// SIMATIC STEP 7 (V5.x) project L38_X52_EC1
// CPU: CPU
// station: P_ADR_BUS
// station: Matériel
// station: API
// station: P_ADR_BUS
// station: Configuration
// station: MOP
// program: PROG
// program: Programa S7_back

SYMBOL_TABLE
"IBD"	DB 95	DB 95	// FACILITY: DATA BASE DB / DB BASE DE DONNEE
"IIT"	DB 96	DB 96	// FACILITY: PART TABLE / DB TABLE PIECE
END_SYMBOL_TABLE

DATA_BLOCK "IBD"	// DB 95
TITLE = FACILITY: DATABASE DB CONTROL
NAME : IBD
VERSION : 0.1
  STRUCT
   BDD : ARRAY  [1 .. 8, 1 .. 200 ] OF WORD ;	//SPARE
  END_STRUCT ;	
BEGIN
END_DATA_BLOCK

DATA_BLOCK "IIT"	// DB 96
TITLE = FACILITY: PART WORD TABLE
NAME : IIT
VERSION : 1.0
  STRUCT
   A0 : STRUCT 	//PART WORD A0
    MP : STRUCT 	//PART MEMORY / MOT PIECE
     MPP : BOOL ;	//PRESENT PART MEMORY / MEMOIRE PIECE PRESENTE
     MPAT : BOOL ;	//PART WITH WORK MEMORY / MEMOIRE PIECE A TRAVAILLER
     MPST : BOOL ;	//PART WITHOUT WORK MEMORY / MEMOIRE PIECE SANS TRAVAIL
     MPAM : BOOL ;	//PART MEMORY TO MATCH / MEMOIRE PIECE A MARIER
     MPAE : BOOL ;	//PART MEMORY TO EVACUATE / MEMOIRE PIECE A EVACUER
     MPP1 : BOOL ;	//INTERMEDIATE PRESENT PART MEMORY / MEMOIRE PIECE PRESENTE INTERMEDIAIRE
     MPP2 : BOOL ;	//INTERMEDIATE PRESENT PART MEMORY / MEMOIRE PIECE PRESENTE INTERMEDIAIRE
     MPP3 : BOOL ;	//INTERMEDIATE PRESENT PART MEMORY / MEMOIRE PIECE PRESENTE INTERMEDIAIRE
     MPP4 : BOOL ;	//INTERMEDIATE PRESENT PART MEMORY / MEMOIRE PIECE PRESENTE INTERMEDIAIRE
     MPP5 : BOOL ;	//INTERMEDIATE PRESENT PART MEMORY / MEMOIRE PIECE PRESENTE INTERMEDIAIRE
     MPP6 : BOOL ;	//INTERMEDIATE PRESENT PART MEMORY / MEMOIRE PIECE PRESENTE INTERMEDIAIRE
     MPP7 : BOOL ;	//INTERMEDIATE PRESENT PART MEMORY / MEMOIRE PIECE PRESENTE INTERMEDIAIRE
     MPP8 : BOOL ;	//INTERMEDIATE PRESENT PART MEMORY / MEMOIRE PIECE PRESENTE INTERMEDIAIRE
     MPT : BOOL ;	//PART COMPLETE MEMORY / MEMOIRE PIECE TRAVAILLE
     MPLNOK : BOOL ;	//LAUCHING PART MEMORY NOK / MEMOIRE LANCEMENT PIECE NON OK
     MPLNOR : BOOL ;	//LAUCHING PART MEMORY OK / MEMOIRE LANCEMENT PIECE OK
    END_STRUCT ;
    MS : STRUCT 	//SUPPORT WORD / MOT SUPPORT
     MSP : BOOL ;	//SUPPORT PRESENCE MEMORY / MEMOIRE SUPPORT PRESENT
     MSAE : BOOL ;	//SUPPORT TO EVACUATE MEMORY / MEMOIRE SUPPORT A EVACUER
     MSEBD : BOOL ;	//WRITING DATABASE SUPPORT MEMORY / MEMOIRE SUPPORT ECRITURE BASE DE DONNEE
     MSMBD : BOOL ;	//MODIFICATION DATABASE SUPPORT MEMORY / MEMOIRE SUPPORT MODIF BASE DE DONNEE
     MSLBD : BOOL ;	//READING DATABASE SUPPORT MEMORY / MEMOIRE SUPPORT LECTURE BASE DE DONNEE
     MSAP : BOOL ;	//PASSAGE AUTHORIZATION SUPPORT MEMORY / MEMOIRE SUPPORT AUTORISATION DE PASSAGE
     MRCPF : BOOL ;	//PART TO DO PROCESS CODE SEARCH MEMORY / MEMOIRE RECH CODES PROCESS A FAIRE
     MRCPS : BOOL ;	//NEXT PART PROCESS CODE SEARCH MEMORY / MEMOIRE RECH CODES PROCESS SUIVANT
     MSLRFID : BOOL ;	//READING RFID SUPPORT MEMORY / MEMOIRE SUPPORT LECTURE RFID
     MSERFID : BOOL ;	//WRITING RFID SUPPORT MEMORY / MEMOIRE SUPPORT ECRITURE RFID
     RES1 : BOOL ;	//SPARE / RESERVE
     RES2 : BOOL ;	//SPARE / RESERVE
     RES3 : BOOL ;	//SPARE / RESERVE
     RES4 : BOOL ;	//SPARE / RESERVE
     RES5 : BOOL ;	//SPARE / RESERVE
     MSLHS : BOOL ;	//LOCAL PRODUCTION MEMORY SUPPORT / MEMOIRE SUPPORT LANCE HORS SIPTOL
    END_STRUCT ;
    NSUP : INT ;	//SUPPORT NUMBER / NUMERO DE SUPPORT
    NFILM : INT ;	//FILM NUMBER / NUMERO DE FILM
    NORDRE : INT ;	//ORDER NUMBER / NUMERO D ORDRE
    CDIV1 : INT ;	//FAMILIA / FAMILLE (CDIV1)
    CDIV2 : INT ;	//FASE / PHASE (CDIV2)
    CDIV3 : INT ;	//MODELO / MODELE (CDIV3)
    CDIV4 : INT ;	//TECHO (CDIV4)
    CDIV5 : INT ;	//VERSION (CDIV5)
    DESFI : INT ;	//FINAL DISPATCH / DESTINATION FINALE
    CSORT : INT ;	//CAUSE DE SORTIE
    DAT : STRUCT 	//DEFINITION / ATTENTE TRAVAIL
     B8 : BOOL ;	//PALETTE DE VIDAGE PERIMETRE (HORS SIPTOL)
     B9 : BOOL ;	//DEVERMINAGE PIECE / PALETTE (HORS SIPTOL)
     B10 : BOOL ;	//PALETTE DE MAP(HORS SIPTOL)
     B11 : BOOL ;	//PALETTE DE CHANGEMENT ELECTRODE BR (HORS SIPTOL)
     B12 : BOOL ;	//PALETTE DE CHANGEMENT ELECTRODE CS (HORS SIPTOL)
     B13 : BOOL ;	//DEVERMINAGE PIECE / PALETTE (AVEC SIPTOL)
     B14 : BOOL ;
     B15 : BOOL ;
     FABSPF : BOOL ;	//0 = AVEC TRAVAIL / 1 = SANS TRAVAIL (P1)
     B1 : BOOL ;
     B2 : BOOL ;	//0 = SUPPORT PLEIN / 1 = SUPPORT VIDE
     B3 : BOOL ;
     B4 : BOOL ;
     B5 : BOOL ;
     B6 : BOOL ;
     B7 : BOOL ;
    END_STRUCT ;
    CRAPI : STRUCT 	//PLC DISPATCHING REASON / CAUSE ROUTAGE API
     B8 : BOOL ;
     B9 : BOOL ;
     B10 : BOOL ;
     B11 : BOOL ;
     B12 : BOOL ;
     B13 : BOOL ;
     B14 : BOOL ;
     B15 : BOOL ;
     B0 : BOOL ;
     B1 : BOOL ;
     B2 : BOOL ;
     RARET : BOOL ;	//PIECE ANALYSE - RETOUCHE
     B4 : BOOL ;
     B5 : BOOL ;
     B6 : BOOL ;
     B7 : BOOL ;
    END_STRUCT ;
    MGEST : STRUCT 	//MOT DE GESTION RECALAGE
     MPFNOR : BOOL ;	//MEMOIRE PIECE FLUX NORMAL
     MPSTC : BOOL ;	//MEMOIRE PIECE A SORTIR TOUS CAS
     MPSOR : BOOL ;	//MEMOIRE PIECE A SORTIR (SORTIE SIPTOL BONNE)
     MPSSU : BOOL ;	//MEMOIRE PIECE A SORTIR (SUBTITUTION PIECE BONNE)
     MPSDI : BOOL ;	//MEMOIRE PIECE A SORTIR (DISCORDANCE)
     MPSSUL : BOOL ;	//MEMOIRE PIECE A SORTIR (SUBTITUTION PIECE LOUPEE)
     MPSL : BOOL ;	//MEMOIRE PIECE A SORTIR (SORTIE LOUPEE)
     MPSF99 : BOOL ;	//MEMOIRE PIECE A SORTIR (MAP FILM 99)
     MPETC : BOOL ;	//MEMOIRE PIECE A ENTRER TOUTS CAS
     MPEOR : BOOL ;	//MEMOIRE PIECE EN ENTREE (DEMANDE SIPTOL)
     MPESUB : BOOL ;	//MEMOIRE PIECE EN ENTREE (SUBTITUTION PIECE BONNE)
     MPEDI : BOOL ;	//MEMOIRE PIECE EN ENTREE (DISCORDANCE)
     MPESUL : BOOL ;	//MEMOIRE PIECE EN ENTREE (SUBTITUTION PIECE LOUPEE)
     MPOCV : BOOL ;	//MEMOIRE PIECE A SORTIR VEHICULE ANNULE + CROCHET VIDE
     MESUTC : BOOL ;	//MEMOIRE EN ENTREE SUBSTITUTION TOUS CAS (PIECE BONNE OU MAUVAISE)
     MSSUTC : BOOL ;	//MEMOIRE SORTIE SUBSTITUTION TOUS CAS (PIECE BONNE OU MAUVAISE)
    END_STRUCT ;
    TVEH : STRUCT 	//TYPO DE VEHICULO
     B8 : BOOL ;
     B9 : BOOL ;
     B10 : BOOL ;
     B11 : BOOL ;
     B12 : BOOL ;
     B13 : BOOL ;
     B14 : BOOL ;
     FABSPF : BOOL ;	//FABRICATION SANS PIECE AU FILM
     SPE : BOOL ;	//UNIT ESPECIAL
     B1 : BOOL ;
     B2 : BOOL ;
     B3 : BOOL ;
     B4 : BOOL ;
     B5 : BOOL ;
     B6 : BOOL ;
     B7 : BOOL ;
    END_STRUCT ;
    SPARE : ARRAY  [1 .. 4 ] OF INT ;	//SPARE
   END_STRUCT ;
   A0_TT : STRUCT 	//WORK TABLE A0
    MFT : STRUCT 	//END OF WORK MEMORY
     MFT1 : BOOL ;	//END OF WORK MEMORY 1 - SPARE
     MFT2 : BOOL ;	//END OF WORK MEMORY 2 - SPARE
     MFT3 : BOOL ;	//END OF WORK MEMORY 3 - SPARE
     MFT4 : BOOL ;	//END OF WORK MEMORY 4 - SPARE
     MFT5 : BOOL ;	//END OF WORK MEMORY 5 - SPARE
     MFT6 : BOOL ;	//END OF WORK MEMORY 6 - SPARE
     MFT7 : BOOL ;	//END OF WORK MEMORY 7 - SPARE
     MFT8 : BOOL ;	//END OF WORK MEMORY 8 - SPARE
     MFT9 : BOOL ;	//END OF WORK MEMORY 9 - SPARE
     MFT10 : BOOL ;	//END OF WORK MEMORY 10 - SPARE
     MFT11 : BOOL ;	//END OF WORK MEMORY 11 - SPARE
     MFT12 : BOOL ;	//END OF WORK MEMORY 12 - SPARE
     MFT13 : BOOL ;	//END OF WORK MEMORY 13 - SPARE
     MFT14 : BOOL ;	//END OF WORK MEMORY 14 - SPARE
     MFT15 : BOOL ;	//END OF WORK MEMORY 15 - SPARE
     MFT16 : BOOL ;	//END OF WORK MEMORY 16 - SPARE
    END_STRUCT ;
    A1 : STRUCT 	//END OF WORK MEMORY A1
     MFT1 : BOOL ;	//END OF WORK MEMORY 1 - SPARE
     MFT2 : BOOL ;	//END OF WORK MEMORY 2 - SPARE
     MFT3 : BOOL ;	//END OF WORK MEMORY 3 - SPARE
     MFT4 : BOOL ;	//END OF WORK MEMORY 4 - SPARE
     MFT5 : BOOL ;	//END OF WORK MEMORY 5 - SPARE
     MFT6 : BOOL ;	//END OF WORK MEMORY 6 - SPARE
     MFT7 : BOOL ;	//END OF WORK MEMORY 7 - SPARE
     MFT8 : BOOL ;	//END OF WORK MEMORY 8 - SPARE
    END_STRUCT ;
    A2 : STRUCT 	//END OF WORK MEMORY A2
     MFT1 : BOOL ;	//END OF WORK MEMORY 1 - SPARE
     MFT2 : BOOL ;	//END OF WORK MEMORY 2 - SPARE
     MFT3 : BOOL ;	//END OF WORK MEMORY 3 - SPARE
     MFT4 : BOOL ;	//END OF WORK MEMORY 4 - SPARE
     MFT5 : BOOL ;	//END OF WORK MEMORY 5 - SPARE
     MFT6 : BOOL ;	//END OF WORK MEMORY 6 - SPARE
     MFT7 : BOOL ;	//END OF WORK MEMORY 7 - SPARE
     MFT8 : BOOL ;	//END OF WORK MEMORY 8 - SPARE
    END_STRUCT ;
    A3 : STRUCT 	//END OF WORK MEMORY A3
     MFT1 : BOOL ;	//END OF WORK MEMORY 1 - SPARE
     MFT2 : BOOL ;	//END OF WORK MEMORY 2 - SPARE
     MFT3 : BOOL ;	//END OF WORK MEMORY 3 - SPARE
     MFT4 : BOOL ;	//END OF WORK MEMORY 4 - SPARE
     MFT5 : BOOL ;	//END OF WORK MEMORY 5 - SPARE
     MFT6 : BOOL ;	//END OF WORK MEMORY 6 - SPARE
     MFT7 : BOOL ;	//END OF WORK MEMORY 7 - SPARE
     MFT8 : BOOL ;	//END OF WORK MEMORY 8 - SPARE
    END_STRUCT ;
    SPARE : ARRAY  [1 .. 16 ] OF INT ;	//SPARE
   END_STRUCT ;
   A0w : STRUCT 	//PART WORD A0w
    MP : STRUCT 	//PART MEMORY / MOT PIECE
     MPP : BOOL ;	//PRESENT PART MEMORY / MEMOIRE PIECE PRESENTE
     MPAT : BOOL ;	//PART WITH WORK MEMORY / MEMOIRE PIECE A TRAVAILLER
     MPST : BOOL ;	//PART WITHOUT WORK MEMORY / MEMOIRE PIECE SANS TRAVAIL
     MPAM : BOOL ;	//PART MEMORY TO MATCH / MEMOIRE PIECE A MARIER
     MPAE : BOOL ;	//PART MEMORY TO EVACUATE / MEMOIRE PIECE A EVACUER
     MPP1 : BOOL ;	//INTERMEDIATE PRESENT PART MEMORY / MEMOIRE PIECE PRESENTE INTERMEDIAIRE
     MPP2 : BOOL ;	//INTERMEDIATE PRESENT PART MEMORY / MEMOIRE PIECE PRESENTE INTERMEDIAIRE
     MPP3 : BOOL ;	//INTERMEDIATE PRESENT PART MEMORY / MEMOIRE PIECE PRESENTE INTERMEDIAIRE
     MPP4 : BOOL ;	//INTERMEDIATE PRESENT PART MEMORY / MEMOIRE PIECE PRESENTE INTERMEDIAIRE
     MPP5 : BOOL ;	//INTERMEDIATE PRESENT PART MEMORY / MEMOIRE PIECE PRESENTE INTERMEDIAIRE
     MPP6 : BOOL ;	//INTERMEDIATE PRESENT PART MEMORY / MEMOIRE PIECE PRESENTE INTERMEDIAIRE
     MPP7 : BOOL ;	//INTERMEDIATE PRESENT PART MEMORY / MEMOIRE PIECE PRESENTE INTERMEDIAIRE
     MPP8 : BOOL ;	//INTERMEDIATE PRESENT PART MEMORY / MEMOIRE PIECE PRESENTE INTERMEDIAIRE
     MPT : BOOL ;	//PART COMPLETE MEMORY / MEMOIRE PIECE TRAVAILLE
     MPLNOK : BOOL ;	//LAUCHING PART MEMORY NOK / MEMOIRE LANCEMENT PIECE NON OK
     MPLNOR : BOOL ;	//LAUCHING PART MEMORY OK / MEMOIRE LANCEMENT PIECE OK
    END_STRUCT ;
    MS : STRUCT 	//SUPPORT WORD / MOT SUPPORT
     MSP : BOOL ;	//SUPPORT PRESENCE MEMORY / MEMOIRE SUPPORT PRESENT
     MSAE : BOOL ;	//SUPPORT TO EVACUATE MEMORY / MEMOIRE SUPPORT A EVACUER
     MSEBD : BOOL ;	//WRITING DATABASE SUPPORT MEMORY / MEMOIRE SUPPORT ECRITURE BASE DE DONNEE
     MSMBD : BOOL ;	//MODIFICATION DATABASE SUPPORT MEMORY / MEMOIRE SUPPORT MODIF BASE DE DONNEE
     MSLBD : BOOL ;	//READING DATABASE SUPPORT MEMORY / MEMOIRE SUPPORT LECTURE BASE DE DONNEE
     MSAP : BOOL ;	//PASSAGE AUTHORIZATION SUPPORT MEMORY / MEMOIRE SUPPORT AUTORISATION DE PASSAGE
     MRCPF : BOOL ;	//PART TO DO PROCESS CODE SEARCH MEMORY / MEMOIRE RECH CODES PROCESS A FAIRE
     MRCPS : BOOL ;	//NEXT PART PROCESS CODE SEARCH MEMORY / MEMOIRE RECH CODES PROCESS SUIVANT
     MSLRFID : BOOL ;	//READING RFID SUPPORT MEMORY / MEMOIRE SUPPORT LECTURE RFID
     MSERFID : BOOL ;	//WRITING RFID SUPPORT MEMORY / MEMOIRE SUPPORT ECRITURE RFID
     RES1 : BOOL ;	//SPARE / RESERVE
     RES2 : BOOL ;	//SPARE / RESERVE
     RES3 : BOOL ;	//SPARE / RESERVE
     RES4 : BOOL ;	//SPARE / RESERVE
     RES5 : BOOL ;	//SPARE / RESERVE
     RES6 : BOOL ;	//SPARE / RESERVE
    END_STRUCT ;
    NSUP : INT ;	//SUPPORT NUMBER / NUMERO DE SUPPORT
    NFILM : INT ;	//FILM NUMBER / NUMERO DE FILM
    NORDRE : INT ;	//ORDER NUMBER / NUMERO D ORDRE
    CDIV1 : INT ;	//FAMILIA / FAMILLE (CDIV1)
    CDIV2 : INT ;	//FASE / PHASE (CDIV2)
    CDIV3 : INT ;	//MODELO / MODELE (CDIV3)
    CDIV4 : INT ;	//TECHO (CDIV4)
    CDIV5 : INT ;	//VERSION (CDIV5)
    DESFI : INT ;	//FINAL DISPATCH / DESTINATION FINALE
    CSORT : INT ;	//CAUSE DE SORTIE
    DAT : STRUCT 	//DEFINITION / ATTENTE TRAVAIL
     B8 : BOOL ;	//PALETTE DE VIDAGE PERIMETRE (HORS SIPTOL)
     B9 : BOOL ;	//DEVERMINAGE PIECE / PALETTE (HORS SIPTOL)
     B10 : BOOL ;	//PALETTE DE MAP(HORS SIPTOL)
     B11 : BOOL ;	//PALETTE DE CHANGEMENT ELECTRODE BR (HORS SIPTOL)
     B12 : BOOL ;	//PALETTE DE CHANGEMENT ELECTRODE CS (HORS SIPTOL)
     B13 : BOOL ;	//DEVERMINAGE PIECE / PALETTE (AVEC SIPTOL)
     B14 : BOOL ;
     B15 : BOOL ;
     FABSPF : BOOL ;	//0 = AVEC TRAVAIL / 1 = SANS TRAVAIL (P1)
     B1 : BOOL ;
     B2 : BOOL ;	//0 = SUPPORT PLEIN / 1 = SUPPORT VIDE
     B3 : BOOL ;
     B4 : BOOL ;
     B5 : BOOL ;
     B6 : BOOL ;
     B7 : BOOL ;
    END_STRUCT ;
    CRAPI : STRUCT 	//PLC DISPATCHING REASON / CAUSE ROUTAGE API
     B8 : BOOL ;
     B9 : BOOL ;
     B10 : BOOL ;
     B11 : BOOL ;
     B12 : BOOL ;
     B13 : BOOL ;
     B14 : BOOL ;
     B15 : BOOL ;
     B0 : BOOL ;
     B1 : BOOL ;
     B2 : BOOL ;
     RARET : BOOL ;	//PIECE ANALYSE - RETOUCHE
     B4 : BOOL ;
     B5 : BOOL ;
     B6 : BOOL ;
     B7 : BOOL ;
    END_STRUCT ;
    MGEST : STRUCT 	//MOT DE GESTION RECALAGE
     MPFNOR : BOOL ;	//MEMOIRE PIECE FLUX NORMAL
     MPSTC : BOOL ;	//MEMOIRE PIECE A SORTIR TOUS CAS
     MPSOR : BOOL ;	//MEMOIRE PIECE A SORTIR (SORTIE SIPTOL BONNE)
     MPSSU : BOOL ;	//MEMOIRE PIECE A SORTIR (SUBTITUTION PIECE BONNE)
     MPSDI : BOOL ;	//MEMOIRE PIECE A SORTIR (DISCORDANCE)
     MPSSUL : BOOL ;	//MEMOIRE PIECE A SORTIR (SUBTITUTION PIECE LOUPEE)
     MPSL : BOOL ;	//MEMOIRE PIECE A SORTIR (SORTIE LOUPEE)
     MPSF99 : BOOL ;	//MEMOIRE PIECE A SORTIR (MAP FILM 99)
     MPETC : BOOL ;	//MEMOIRE PIECE A ENTRER TOUTS CAS
     MPEOR : BOOL ;	//MEMOIRE PIECE EN ENTREE (DEMANDE SIPTOL)
     MPESUB : BOOL ;	//MEMOIRE PIECE EN ENTREE (SUBTITUTION PIECE BONNE)
     MPEDI : BOOL ;	//MEMOIRE PIECE EN ENTREE (DISCORDANCE)
     MPESUL : BOOL ;	//MEMOIRE PIECE EN ENTREE (SUBTITUTION PIECE LOUPEE)
     MPOCV : BOOL ;	//MEMOIRE PIECE A SORTIR VEHICULE ANNULE + CROCHET VIDE
     MESUTC : BOOL ;	//MEMOIRE EN ENTREE SUBSTITUTION TOUS CAS (PIECE BONNE OU MAUVAISE)
     MSSUTC : BOOL ;	//MEMOIRE SORTIE SUBSTITUTION TOUS CAS (PIECE BONNE OU MAUVAISE)
    END_STRUCT ;
    TVEH : STRUCT 	//TYPO DE VEHICULO
     B8 : BOOL ;
     B9 : BOOL ;
     B10 : BOOL ;
     B11 : BOOL ;
     B12 : BOOL ;
     B13 : BOOL ;
     B14 : BOOL ;
     FABSPF : BOOL ;	//FABRICATION SANS PIECE AU FILM
     SPE : BOOL ;	//UNIT ESPECIAL
     B1 : BOOL ;
     B2 : BOOL ;
     B3 : BOOL ;
     B4 : BOOL ;
     B5 : BOOL ;
     B6 : BOOL ;
     B7 : BOOL ;
    END_STRUCT ;
    SPARE : ARRAY  [1 .. 4 ] OF INT ;
   END_STRUCT ;
   B0 : STRUCT 	//PART WORD B0
    MP : STRUCT 	//PART MEMORY / MOT PIECE
     MPP : BOOL ;	//PRESENT PART MEMORY / MEMOIRE PIECE PRESENTE
     MPAT : BOOL ;	//PART WITH WORK MEMORY / MEMOIRE PIECE A TRAVAILLER
     MPST : BOOL ;	//PART WITHOUT WORK MEMORY / MEMOIRE PIECE SANS TRAVAIL
     MPAM : BOOL ;	//PART MEMORY TO MATCH / MEMOIRE PIECE A MARIER
     MPAE : BOOL ;	//PART MEMORY TO EVACUATE / MEMOIRE PIECE A EVACUER
     MPP1 : BOOL ;	//INTERMEDIATE PRESENT PART MEMORY / MEMOIRE PIECE PRESENTE INTERMEDIAIRE
     MPP2 : BOOL ;	//INTERMEDIATE PRESENT PART MEMORY / MEMOIRE PIECE PRESENTE INTERMEDIAIRE
     MPP3 : BOOL ;	//INTERMEDIATE PRESENT PART MEMORY / MEMOIRE PIECE PRESENTE INTERMEDIAIRE
     MPP4 : BOOL ;	//INTERMEDIATE PRESENT PART MEMORY / MEMOIRE PIECE PRESENTE INTERMEDIAIRE
     MPP5 : BOOL ;	//INTERMEDIATE PRESENT PART MEMORY / MEMOIRE PIECE PRESENTE INTERMEDIAIRE
     MPP6 : BOOL ;	//INTERMEDIATE PRESENT PART MEMORY / MEMOIRE PIECE PRESENTE INTERMEDIAIRE
     MPP7 : BOOL ;	//INTERMEDIATE PRESENT PART MEMORY / MEMOIRE PIECE PRESENTE INTERMEDIAIRE
     MPP8 : BOOL ;	//INTERMEDIATE PRESENT PART MEMORY / MEMOIRE PIECE PRESENTE INTERMEDIAIRE
     MPT : BOOL ;	//PART COMPLETE MEMORY / MEMOIRE PIECE TRAVAILLE
     MPLNOK : BOOL ;	//LAUCHING PART MEMORY NOK / MEMOIRE LANCEMENT PIECE NON OK
     MPLNOR : BOOL ;	//LAUCHING PART MEMORY OK / MEMOIRE LANCEMENT PIECE OK
    END_STRUCT ;
    MS : STRUCT 	//SUPPORT WORD / MOT SUPPORT
     MSP : BOOL ;	//SUPPORT PRESENCE MEMORY / MEMOIRE SUPPORT PRESENT
     MSAE : BOOL ;	//SUPPORT TO EVACUATE MEMORY / MEMOIRE SUPPORT A EVACUER
     MSEBD : BOOL ;	//WRITING DATABASE SUPPORT MEMORY / MEMOIRE SUPPORT ECRITURE BASE DE DONNEE
     MSMBD : BOOL ;	//MODIFICATION DATABASE SUPPORT MEMORY / MEMOIRE SUPPORT MODIF BASE DE DONNEE
     MSLBD : BOOL ;	//READING DATABASE SUPPORT MEMORY / MEMOIRE SUPPORT LECTURE BASE DE DONNEE
     MSAP : BOOL ;	//PASSAGE AUTHORIZATION SUPPORT MEMORY / MEMOIRE SUPPORT AUTORISATION DE PASSAGE
     MRCPF : BOOL ;	//PART TO DO PROCESS CODE SEARCH MEMORY / MEMOIRE RECH CODES PROCESS A FAIRE
     MRCPS : BOOL ;	//NEXT PART PROCESS CODE SEARCH MEMORY / MEMOIRE RECH CODES PROCESS SUIVANT
     MSLRFID : BOOL ;	//READING RFID SUPPORT MEMORY / MEMOIRE SUPPORT LECTURE RFID
     MSERFID : BOOL ;	//WRITING RFID SUPPORT MEMORY / MEMOIRE SUPPORT ECRITURE RFID
     RES1 : BOOL ;	//SPARE / RESERVE
     RES2 : BOOL ;	//SPARE / RESERVE
     RES3 : BOOL ;	//SPARE / RESERVE
     RES4 : BOOL ;	//SPARE / RESERVE
     RES5 : BOOL ;	//SPARE / RESERVE
     RES6 : BOOL ;	//SPARE / RESERVE
    END_STRUCT ;
    NSUP : INT ;	//SUPPORT NUMBER / NUMERO DE SUPPORT
    NFILM : INT ;	//FILM NUMBER / NUMERO DE FILM
    NORDRE : INT ;	//ORDER NUMBER / NUMERO D ORDRE
    CDIV1 : INT ;	//FAMILIA / FAMILLE (CDIV1)
    CDIV2 : INT ;	//FASE / PHASE (CDIV2)
    CDIV3 : INT ;	//MODELO / MODELE (CDIV3)
    CDIV4 : INT ;	//TECHO (CDIV4)
    CDIV5 : INT ;	//VERSION (CDIV5)
    DESFI : INT ;	//FINAL DISPATCH / DESTINATION FINALE
    CSORT : INT ;	//CAUSE DE SORTIE
    DAT : STRUCT 	//DEFINITION / ATTENTE TRAVAIL
     B8 : BOOL ;	//PALETTE DE VIDAGE PERIMETRE (HORS SIPTOL)
     B9 : BOOL ;	//DEVERMINAGE PIECE / PALETTE (HORS SIPTOL)
     B10 : BOOL ;	//PALETTE DE MAP(HORS SIPTOL)
     B11 : BOOL ;	//PALETTE DE CHANGEMENT ELECTRODE BR (HORS SIPTOL)
     B12 : BOOL ;	//PALETTE DE CHANGEMENT ELECTRODE CS (HORS SIPTOL)
     B13 : BOOL ;	//DEVERMINAGE PIECE / PALETTE (AVEC SIPTOL)
     B14 : BOOL ;
     B15 : BOOL ;
     FABSPF : BOOL ;	//0 = AVEC TRAVAIL / 1 = SANS TRAVAIL (P1)
     B1 : BOOL ;
     B2 : BOOL ;	//0 = SUPPORT PLEIN / 1 = SUPPORT VIDE
     B3 : BOOL ;
     B4 : BOOL ;
     B5 : BOOL ;
     B6 : BOOL ;
     B7 : BOOL ;
    END_STRUCT ;
    CRAPI : STRUCT 	//PLC DISPATCHING REASON / CAUSE ROUTAGE API
     B8 : BOOL ;
     B9 : BOOL ;
     B10 : BOOL ;
     B11 : BOOL ;
     B12 : BOOL ;
     B13 : BOOL ;
     B14 : BOOL ;
     B15 : BOOL ;
     B0 : BOOL ;
     B1 : BOOL ;
     B2 : BOOL ;
     RARET : BOOL ;	//PIECE ANALYSE - RETOUCHE
     B4 : BOOL ;
     B5 : BOOL ;
     B6 : BOOL ;
     B7 : BOOL ;
    END_STRUCT ;
    MGEST : STRUCT 	//MOT DE GESTION RECALAGE
     MPFNOR : BOOL ;	//MEMOIRE PIECE FLUX NORMAL
     MPSTC : BOOL ;	//MEMOIRE PIECE A SORTIR TOUS CAS
     MPSOR : BOOL ;	//MEMOIRE PIECE A SORTIR (SORTIE SIPTOL BONNE)
     MPSSU : BOOL ;	//MEMOIRE PIECE A SORTIR (SUBTITUTION PIECE BONNE)
     MPSDI : BOOL ;	//MEMOIRE PIECE A SORTIR (DISCORDANCE)
     MPSSUL : BOOL ;	//MEMOIRE PIECE A SORTIR (SUBTITUTION PIECE LOUPEE)
     MPSL : BOOL ;	//MEMOIRE PIECE A SORTIR (SORTIE LOUPEE)
     MPSF99 : BOOL ;	//MEMOIRE PIECE A SORTIR (MAP FILM 99)
     MPETC : BOOL ;	//MEMOIRE PIECE A ENTRER TOUTS CAS
     MPEOR : BOOL ;	//MEMOIRE PIECE EN ENTREE (DEMANDE SIPTOL)
     MPESUB : BOOL ;	//MEMOIRE PIECE EN ENTREE (SUBTITUTION PIECE BONNE)
     MPEDI : BOOL ;	//MEMOIRE PIECE EN ENTREE (DISCORDANCE)
     MPESUL : BOOL ;	//MEMOIRE PIECE EN ENTREE (SUBTITUTION PIECE LOUPEE)
     MPOCV : BOOL ;	//MEMOIRE PIECE A SORTIR VEHICULE ANNULE + CROCHET VIDE
     MESUTC : BOOL ;	//MEMOIRE EN ENTREE SUBSTITUTION TOUS CAS (PIECE BONNE OU MAUVAISE)
     MSSUTC : BOOL ;	//MEMOIRE SORTIE SUBSTITUTION TOUS CAS (PIECE BONNE OU MAUVAISE)
    END_STRUCT ;
    TVEH : STRUCT 	//TYPO DE VEHICULO
     B8 : BOOL ;
     B9 : BOOL ;
     B10 : BOOL ;
     B11 : BOOL ;
     B12 : BOOL ;
     B13 : BOOL ;
     B14 : BOOL ;
     FABSPF : BOOL ;	//FABRICATION SANS PIECE AU FILM
     SPE : BOOL ;	//UNIT ESPECIAL
     B1 : BOOL ;
     B2 : BOOL ;
     B3 : BOOL ;
     B4 : BOOL ;
     B5 : BOOL ;
     B6 : BOOL ;
     B7 : BOOL ;
    END_STRUCT ;
    SPARE : ARRAY  [1 .. 4 ] OF INT ;	//SPARE
   END_STRUCT ;
   B0_TT : STRUCT 	//WORK TABLE B0
    MFT : STRUCT 	//END OF WORK MEMORY
     MFT1 : BOOL ;	//END OF WORK MEMORY 1 - SPARE
     MFT2 : BOOL ;	//END OF WORK MEMORY 2 - SPARE
     MFT3 : BOOL ;	//END OF WORK MEMORY 3 - SPARE
     MFT4 : BOOL ;	//END OF WORK MEMORY 4 - SPARE
     MFT5 : BOOL ;	//END OF WORK MEMORY 5 - SPARE
     MFT6 : BOOL ;	//END OF WORK MEMORY 6 - SPARE
     MFT7 : BOOL ;	//END OF WORK MEMORY 7 - SPARE
     MFT8 : BOOL ;	//END OF WORK MEMORY 8 - SPARE
     MFT9 : BOOL ;	//END OF WORK MEMORY 9 - SPARE
     MFT10 : BOOL ;	//END OF WORK MEMORY 10 - SPARE
     MFT11 : BOOL ;	//END OF WORK MEMORY 11 - SPARE
     MFT12 : BOOL ;	//END OF WORK MEMORY 12 - SPARE
     MFT13 : BOOL ;	//END OF WORK MEMORY 13 - SPARE
     MFT14 : BOOL ;	//END OF WORK MEMORY 14 - SPARE
     MFT15 : BOOL ;	//END OF WORK MEMORY 15 - SPARE
     MFT16 : BOOL ;	//END OF WORK MEMORY 16 - SPARE
    END_STRUCT ;
    B1 : STRUCT 	//END OF WORK MEMORY B1
     MFT1 : BOOL ;	//END OF WORK MEMORY 1 - SPARE
     MFT2 : BOOL ;	//END OF WORK MEMORY 2 - SPARE
     MFT3 : BOOL ;	//END OF WORK MEMORY 3 - SPARE
     MFT4 : BOOL ;	//END OF WORK MEMORY 4 - SPARE
     MFT5 : BOOL ;	//END OF WORK MEMORY 5 - SPARE
     MFT6 : BOOL ;	//END OF WORK MEMORY 6 - SPARE
     MFT7 : BOOL ;	//END OF WORK MEMORY 7 - SPARE
     MFT8 : BOOL ;	//END OF WORK MEMORY 8 - SPARE
    END_STRUCT ;
    B2 : STRUCT 	//END OF WORK MEMORY B2
     MFT1 : BOOL ;	//END OF WORK MEMORY 1 - SPARE
     MFT2 : BOOL ;	//END OF WORK MEMORY 2 - SPARE
     MFT3 : BOOL ;	//END OF WORK MEMORY 3 - SPARE
     MFT4 : BOOL ;	//END OF WORK MEMORY 4 - SPARE
     MFT5 : BOOL ;	//END OF WORK MEMORY 5 - SPARE
     MFT6 : BOOL ;	//END OF WORK MEMORY 6 - SPARE
     MFT7 : BOOL ;	//END OF WORK MEMORY 7 - SPARE
     MFT8 : BOOL ;	//END OF WORK MEMORY 8 - SPARE
    END_STRUCT ;
    SPARE : ARRAY  [1 .. 17 ] OF INT ;	//SPARE
   END_STRUCT ;
   B3 : STRUCT 	//PART WORD B0
    MP : STRUCT 	//PART MEMORY / MOT PIECE
     MPP : BOOL ;	//PRESENT PART MEMORY / MEMOIRE PIECE PRESENTE
     MPAT : BOOL ;	//PART WITH WORK MEMORY / MEMOIRE PIECE A TRAVAILLER
     MPST : BOOL ;	//PART WITHOUT WORK MEMORY / MEMOIRE PIECE SANS TRAVAIL
     MPAM : BOOL ;	//PART MEMORY TO MATCH / MEMOIRE PIECE A MARIER
     MPAE : BOOL ;	//PART MEMORY TO EVACUATE / MEMOIRE PIECE A EVACUER
     MPP1 : BOOL ;	//INTERMEDIATE PRESENT PART MEMORY / MEMOIRE PIECE PRESENTE INTERMEDIAIRE
     MPP2 : BOOL ;	//INTERMEDIATE PRESENT PART MEMORY / MEMOIRE PIECE PRESENTE INTERMEDIAIRE
     MPP3 : BOOL ;	//INTERMEDIATE PRESENT PART MEMORY / MEMOIRE PIECE PRESENTE INTERMEDIAIRE
     MPP4 : BOOL ;	//INTERMEDIATE PRESENT PART MEMORY / MEMOIRE PIECE PRESENTE INTERMEDIAIRE
     MPP5 : BOOL ;	//INTERMEDIATE PRESENT PART MEMORY / MEMOIRE PIECE PRESENTE INTERMEDIAIRE
     MPP6 : BOOL ;	//INTERMEDIATE PRESENT PART MEMORY / MEMOIRE PIECE PRESENTE INTERMEDIAIRE
     MPP7 : BOOL ;	//INTERMEDIATE PRESENT PART MEMORY / MEMOIRE PIECE PRESENTE INTERMEDIAIRE
     MPP8 : BOOL ;	//INTERMEDIATE PRESENT PART MEMORY / MEMOIRE PIECE PRESENTE INTERMEDIAIRE
     MPT : BOOL ;	//PART COMPLETE MEMORY / MEMOIRE PIECE TRAVAILLE
     MPLNOK : BOOL ;	//LAUCHING PART MEMORY NOK / MEMOIRE LANCEMENT PIECE NON OK
     MPLNOR : BOOL ;	//LAUCHING PART MEMORY OK / MEMOIRE LANCEMENT PIECE OK
    END_STRUCT ;
    MS : STRUCT 	//SUPPORT WORD / MOT SUPPORT
     MSP : BOOL ;	//SUPPORT PRESENCE MEMORY / MEMOIRE SUPPORT PRESENT
     MSAE : BOOL ;	//SUPPORT TO EVACUATE MEMORY / MEMOIRE SUPPORT A EVACUER
     MSEBD : BOOL ;	//WRITING DATABASE SUPPORT MEMORY / MEMOIRE SUPPORT ECRITURE BASE DE DONNEE
     MSMBD : BOOL ;	//MODIFICATION DATABASE SUPPORT MEMORY / MEMOIRE SUPPORT MODIF BASE DE DONNEE
     MSLBD : BOOL ;	//READING DATABASE SUPPORT MEMORY / MEMOIRE SUPPORT LECTURE BASE DE DONNEE
     MSAP : BOOL ;	//PASSAGE AUTHORIZATION SUPPORT MEMORY / MEMOIRE SUPPORT AUTORISATION DE PASSAGE
     MRCPF : BOOL ;	//PART TO DO PROCESS CODE SEARCH MEMORY / MEMOIRE RECH CODES PROCESS A FAIRE
     MRCPS : BOOL ;	//NEXT PART PROCESS CODE SEARCH MEMORY / MEMOIRE RECH CODES PROCESS SUIVANT
     MSLRFID : BOOL ;	//READING RFID SUPPORT MEMORY / MEMOIRE SUPPORT LECTURE RFID
     MSERFID : BOOL ;	//WRITING RFID SUPPORT MEMORY / MEMOIRE SUPPORT ECRITURE RFID
     RES1 : BOOL ;	//SPARE / RESERVE
     RES2 : BOOL ;	//SPARE / RESERVE
     RES3 : BOOL ;	//SPARE / RESERVE
     RES4 : BOOL ;	//SPARE / RESERVE
     RES5 : BOOL ;	//SPARE / RESERVE
     RES6 : BOOL ;	//SPARE / RESERVE
    END_STRUCT ;
    NSUP : INT ;	//SUPPORT NUMBER / NUMERO DE SUPPORT
    NFILM : INT ;	//FILM NUMBER / NUMERO DE FILM
    NORDRE : INT ;	//ORDER NUMBER / NUMERO D ORDRE
    CDIV1 : INT ;	//FAMILIA / FAMILLE (CDIV1)
    CDIV2 : INT ;	//FASE / PHASE (CDIV2)
    CDIV3 : INT ;	//MODELO / MODELE (CDIV3)
    CDIV4 : INT ;	//TECHO (CDIV4)
    CDIV5 : INT ;	//VERSION (CDIV5)
    DESFI : INT ;	//FINAL DISPATCH / DESTINATION FINALE
    CSORT : INT ;	//CAUSE DE SORTIE
    DAT : STRUCT 	//DEFINITION / ATTENTE TRAVAIL
     B8 : BOOL ;	//PALETTE DE VIDAGE PERIMETRE (HORS SIPTOL)
     B9 : BOOL ;	//DEVERMINAGE PIECE / PALETTE (HORS SIPTOL)
     B10 : BOOL ;	//PALETTE DE MAP(HORS SIPTOL)
     B11 : BOOL ;	//PALETTE DE CHANGEMENT ELECTRODE BR (HORS SIPTOL)
     B12 : BOOL ;	//PALETTE DE CHANGEMENT ELECTRODE CS (HORS SIPTOL)
     B13 : BOOL ;	//DEVERMINAGE PIECE / PALETTE (AVEC SIPTOL)
     B14 : BOOL ;
     B15 : BOOL ;
     FABSPF : BOOL ;	//0 = AVEC TRAVAIL / 1 = SANS TRAVAIL (P1)
     B1 : BOOL ;
     B2 : BOOL ;	//0 = SUPPORT PLEIN / 1 = SUPPORT VIDE
     B3 : BOOL ;
     B4 : BOOL ;
     B5 : BOOL ;
     B6 : BOOL ;
     B7 : BOOL ;
    END_STRUCT ;
    CRAPI : STRUCT 	//PLC DISPATCHING REASON / CAUSE ROUTAGE API
     B8 : BOOL ;
     B9 : BOOL ;
     B10 : BOOL ;
     B11 : BOOL ;
     B12 : BOOL ;
     B13 : BOOL ;
     B14 : BOOL ;
     B15 : BOOL ;
     B0 : BOOL ;
     B1 : BOOL ;
     B2 : BOOL ;
     RARET : BOOL ;	//PIECE ANALYSE - RETOUCHE
     B4 : BOOL ;
     B5 : BOOL ;
     B6 : BOOL ;
     B7 : BOOL ;
    END_STRUCT ;
    MGEST : STRUCT 	//MOT DE GESTION RECALAGE
     MPFNOR : BOOL ;	//MEMOIRE PIECE FLUX NORMAL
     MPSTC : BOOL ;	//MEMOIRE PIECE A SORTIR TOUS CAS
     MPSOR : BOOL ;	//MEMOIRE PIECE A SORTIR (SORTIE SIPTOL BONNE)
     MPSSU : BOOL ;	//MEMOIRE PIECE A SORTIR (SUBTITUTION PIECE BONNE)
     MPSDI : BOOL ;	//MEMOIRE PIECE A SORTIR (DISCORDANCE)
     MPSSUL : BOOL ;	//MEMOIRE PIECE A SORTIR (SUBTITUTION PIECE LOUPEE)
     MPSL : BOOL ;	//MEMOIRE PIECE A SORTIR (SORTIE LOUPEE)
     MPSF99 : BOOL ;	//MEMOIRE PIECE A SORTIR (MAP FILM 99)
     MPETC : BOOL ;	//MEMOIRE PIECE A ENTRER TOUTS CAS
     MPEOR : BOOL ;	//MEMOIRE PIECE EN ENTREE (DEMANDE SIPTOL)
     MPESUB : BOOL ;	//MEMOIRE PIECE EN ENTREE (SUBTITUTION PIECE BONNE)
     MPEDI : BOOL ;	//MEMOIRE PIECE EN ENTREE (DISCORDANCE)
     MPESUL : BOOL ;	//MEMOIRE PIECE EN ENTREE (SUBTITUTION PIECE LOUPEE)
     MPOCV : BOOL ;	//MEMOIRE PIECE A SORTIR VEHICULE ANNULE + CROCHET VIDE
     MESUTC : BOOL ;	//MEMOIRE EN ENTREE SUBSTITUTION TOUS CAS (PIECE BONNE OU MAUVAISE)
     MSSUTC : BOOL ;	//MEMOIRE SORTIE SUBSTITUTION TOUS CAS (PIECE BONNE OU MAUVAISE)
    END_STRUCT ;
    SPARE : ARRAY  [1 .. 5 ] OF INT ;
   END_STRUCT ;
   B3_TT : STRUCT 	//WORK TABLE B0
    MFT : STRUCT 	//END OF WORK MEMORY
     MFT1 : BOOL ;	//END OF WORK MEMORY 1 - SPARE
     MFT2 : BOOL ;	//END OF WORK MEMORY 2 - SPARE
     MFT3 : BOOL ;	//END OF WORK MEMORY 3 - SPARE
     MFT4 : BOOL ;	//END OF WORK MEMORY 4 - SPARE
     MFT5 : BOOL ;	//END OF WORK MEMORY 5 - SPARE
     MFT6 : BOOL ;	//END OF WORK MEMORY 6 - SPARE
     MFT7 : BOOL ;	//END OF WORK MEMORY 7 - SPARE
     MFT8 : BOOL ;	//END OF WORK MEMORY 8 - SPARE
     MFT9 : BOOL ;	//END OF WORK MEMORY 9 - SPARE
     MFT10 : BOOL ;	//END OF WORK MEMORY 10 - SPARE
     MFT11 : BOOL ;	//END OF WORK MEMORY 11 - SPARE
     MFT12 : BOOL ;	//END OF WORK MEMORY 12 - SPARE
     MFT13 : BOOL ;	//END OF WORK MEMORY 13 - SPARE
     MFT14 : BOOL ;	//END OF WORK MEMORY 14 - SPARE
     MFT15 : BOOL ;	//END OF WORK MEMORY 15 - SPARE
     MFT16 : BOOL ;	//END OF WORK MEMORY 16 - SPARE
    END_STRUCT ;
    B4 : STRUCT 	//END OF WORK MEMORY B1
     MFT1 : BOOL ;	//END OF WORK MEMORY 1 - SPARE
     MFT2 : BOOL ;	//END OF WORK MEMORY 2 - SPARE
     MFT3 : BOOL ;	//END OF WORK MEMORY 3 - SPARE
     MFT4 : BOOL ;	//END OF WORK MEMORY 4 - SPARE
     MFT5 : BOOL ;	//END OF WORK MEMORY 5 - SPARE
     MFT6 : BOOL ;	//END OF WORK MEMORY 6 - SPARE
     MFT7 : BOOL ;	//END OF WORK MEMORY 7 - SPARE
     MFT8 : BOOL ;	//END OF WORK MEMORY 8 - SPARE
    END_STRUCT ;
    B5 : STRUCT 	//END OF WORK MEMORY B2
     MFT1 : BOOL ;	//END OF WORK MEMORY 1 - SPARE
     MFT2 : BOOL ;	//END OF WORK MEMORY 2 - SPARE
     MFT3 : BOOL ;	//END OF WORK MEMORY 3 - SPARE
     MFT4 : BOOL ;	//END OF WORK MEMORY 4 - SPARE
     MFT5 : BOOL ;	//END OF WORK MEMORY 5 - SPARE
     MFT6 : BOOL ;	//END OF WORK MEMORY 6 - SPARE
     MFT7 : BOOL ;	//END OF WORK MEMORY 7 - SPARE
     MFT8 : BOOL ;	//END OF WORK MEMORY 8 - SPARE
     SPARE : ARRAY  [1 .. 3 ] OF INT ;
    END_STRUCT ;
   END_STRUCT ;
   B0w : STRUCT 	//PART WORD B0w
    MP : STRUCT 	//PART MEMORY / MOT PIECE
     MPP : BOOL ;	//PRESENT PART MEMORY / MEMOIRE PIECE PRESENTE
     MPAT : BOOL ;	//PART WITH WORK MEMORY / MEMOIRE PIECE A TRAVAILLER
     MPST : BOOL ;	//PART WITHOUT WORK MEMORY / MEMOIRE PIECE SANS TRAVAIL
     MPAM : BOOL ;	//PART MEMORY TO MATCH / MEMOIRE PIECE A MARIER
     MPAE : BOOL ;	//PART MEMORY TO EVACUATE / MEMOIRE PIECE A EVACUER
     MPP1 : BOOL ;	//INTERMEDIATE PRESENT PART MEMORY / MEMOIRE PIECE PRESENTE INTERMEDIAIRE
     MPP2 : BOOL ;	//INTERMEDIATE PRESENT PART MEMORY / MEMOIRE PIECE PRESENTE INTERMEDIAIRE
     MPP3 : BOOL ;	//INTERMEDIATE PRESENT PART MEMORY / MEMOIRE PIECE PRESENTE INTERMEDIAIRE
     MPP4 : BOOL ;	//INTERMEDIATE PRESENT PART MEMORY / MEMOIRE PIECE PRESENTE INTERMEDIAIRE
     MPP5 : BOOL ;	//INTERMEDIATE PRESENT PART MEMORY / MEMOIRE PIECE PRESENTE INTERMEDIAIRE
     MPP6 : BOOL ;	//INTERMEDIATE PRESENT PART MEMORY / MEMOIRE PIECE PRESENTE INTERMEDIAIRE
     MPP7 : BOOL ;	//INTERMEDIATE PRESENT PART MEMORY / MEMOIRE PIECE PRESENTE INTERMEDIAIRE
     MPP8 : BOOL ;	//INTERMEDIATE PRESENT PART MEMORY / MEMOIRE PIECE PRESENTE INTERMEDIAIRE
     MPT : BOOL ;	//PART COMPLETE MEMORY / MEMOIRE PIECE TRAVAILLE
     MPLNOK : BOOL ;	//LAUCHING PART MEMORY NOK / MEMOIRE LANCEMENT PIECE NON OK
     MPLNOR : BOOL ;	//LAUCHING PART MEMORY OK / MEMOIRE LANCEMENT PIECE OK
    END_STRUCT ;
    MS : STRUCT 	//SUPPORT WORD / MOT SUPPORT
     MSP : BOOL ;	//SUPPORT PRESENCE MEMORY / MEMOIRE SUPPORT PRESENT
     MSAE : BOOL ;	//SUPPORT TO EVACUATE MEMORY / MEMOIRE SUPPORT A EVACUER
     MSEBD : BOOL ;	//WRITING DATABASE SUPPORT MEMORY / MEMOIRE SUPPORT ECRITURE BASE DE DONNEE
     MSMBD : BOOL ;	//MODIFICATION DATABASE SUPPORT MEMORY / MEMOIRE SUPPORT MODIF BASE DE DONNEE
     MSLBD : BOOL ;	//READING DATABASE SUPPORT MEMORY / MEMOIRE SUPPORT LECTURE BASE DE DONNEE
     MSAP : BOOL ;	//PASSAGE AUTHORIZATION SUPPORT MEMORY / MEMOIRE SUPPORT AUTORISATION DE PASSAGE
     MRCPF : BOOL ;	//PART TO DO PROCESS CODE SEARCH MEMORY / MEMOIRE RECH CODES PROCESS A FAIRE
     MRCPS : BOOL ;	//NEXT PART PROCESS CODE SEARCH MEMORY / MEMOIRE RECH CODES PROCESS SUIVANT
     MSLRFID : BOOL ;	//READING RFID SUPPORT MEMORY / MEMOIRE SUPPORT LECTURE RFID
     MSERFID : BOOL ;	//WRITING RFID SUPPORT MEMORY / MEMOIRE SUPPORT ECRITURE RFID
     RES1 : BOOL ;	//SPARE / RESERVE
     RES2 : BOOL ;	//SPARE / RESERVE
     RES3 : BOOL ;	//SPARE / RESERVE
     RES4 : BOOL ;	//SPARE / RESERVE
     RES5 : BOOL ;	//SPARE / RESERVE
     RES6 : BOOL ;	//SPARE / RESERVE
    END_STRUCT ;
    NSUP : INT ;	//SUPPORT NUMBER / NUMERO DE SUPPORT
    NFILM : INT ;	//FILM NUMBER / NUMERO DE FILM
    NORDRE : INT ;	//ORDER NUMBER / NUMERO D ORDRE
    CDIV1 : INT ;	//FAMILIA / FAMILLE (CDIV1)
    CDIV2 : INT ;	//FASE / PHASE (CDIV2)
    CDIV3 : INT ;	//MODELO / MODELE (CDIV3)
    CDIV4 : INT ;	//TECHO (CDIV4)
    CDIV5 : INT ;	//VERSION (CDIV5)
    DESFI : INT ;	//FINAL DISPATCH / DESTINATION FINALE
    CSORT : INT ;	//CAUSE DE SORTIE
    DAT : STRUCT 	//DEFINITION / ATTENTE TRAVAIL
     B8 : BOOL ;	//PALETTE DE VIDAGE PERIMETRE (HORS SIPTOL)
     B9 : BOOL ;	//DEVERMINAGE PIECE / PALETTE (HORS SIPTOL)
     B10 : BOOL ;	//PALETTE DE MAP(HORS SIPTOL)
     B11 : BOOL ;	//PALETTE DE CHANGEMENT ELECTRODE BR (HORS SIPTOL)
     B12 : BOOL ;	//PALETTE DE CHANGEMENT ELECTRODE CS (HORS SIPTOL)
     B13 : BOOL ;	//DEVERMINAGE PIECE / PALETTE (AVEC SIPTOL)
     B14 : BOOL ;
     B15 : BOOL ;
     FABSPF : BOOL ;	//0 = AVEC TRAVAIL / 1 = SANS TRAVAIL (P1)
     B1 : BOOL ;
     B2 : BOOL ;	//0 = SUPPORT PLEIN / 1 = SUPPORT VIDE
     B3 : BOOL ;
     B4 : BOOL ;
     B5 : BOOL ;
     B6 : BOOL ;
     B7 : BOOL ;
    END_STRUCT ;
    CRAPI : STRUCT 	//PLC DISPATCHING REASON / CAUSE ROUTAGE API
     B8 : BOOL ;
     B9 : BOOL ;
     B10 : BOOL ;
     B11 : BOOL ;
     B12 : BOOL ;
     B13 : BOOL ;
     B14 : BOOL ;
     B15 : BOOL ;
     B0 : BOOL ;
     B1 : BOOL ;
     B2 : BOOL ;
     RARET : BOOL ;	//PIECE ANALYSE - RETOUCHE
     B4 : BOOL ;
     B5 : BOOL ;
     B6 : BOOL ;
     B7 : BOOL ;
    END_STRUCT ;
    MGEST : STRUCT 	//MOT DE GESTION RECALAGE
     MPFNOR : BOOL ;	//MEMOIRE PIECE FLUX NORMAL
     MPSTC : BOOL ;	//MEMOIRE PIECE A SORTIR TOUS CAS
     MPSOR : BOOL ;	//MEMOIRE PIECE A SORTIR (SORTIE SIPTOL BONNE)
     MPSSU : BOOL ;	//MEMOIRE PIECE A SORTIR (SUBTITUTION PIECE BONNE)
     MPSDI : BOOL ;	//MEMOIRE PIECE A SORTIR (DISCORDANCE)
     MPSSUL : BOOL ;	//MEMOIRE PIECE A SORTIR (SUBTITUTION PIECE LOUPEE)
     MPSL : BOOL ;	//MEMOIRE PIECE A SORTIR (SORTIE LOUPEE)
     MPSF99 : BOOL ;	//MEMOIRE PIECE A SORTIR (MAP FILM 99)
     MPETC : BOOL ;	//MEMOIRE PIECE A ENTRER TOUTS CAS
     MPEOR : BOOL ;	//MEMOIRE PIECE EN ENTREE (DEMANDE SIPTOL)
     MPESUB : BOOL ;	//MEMOIRE PIECE EN ENTREE (SUBTITUTION PIECE BONNE)
     MPEDI : BOOL ;	//MEMOIRE PIECE EN ENTREE (DISCORDANCE)
     MPESUL : BOOL ;	//MEMOIRE PIECE EN ENTREE (SUBTITUTION PIECE LOUPEE)
     MPOCV : BOOL ;	//MEMOIRE PIECE A SORTIR VEHICULE ANNULE + CROCHET VIDE
     MESUTC : BOOL ;	//MEMOIRE EN ENTREE SUBSTITUTION TOUS CAS (PIECE BONNE OU MAUVAISE)
     MSSUTC : BOOL ;	//MEMOIRE SORTIE SUBSTITUTION TOUS CAS (PIECE BONNE OU MAUVAISE)
    END_STRUCT ;
    TVEH : STRUCT 	//TYPO DE VEHICULO
     B8 : BOOL ;
     B9 : BOOL ;
     B10 : BOOL ;
     B11 : BOOL ;
     B12 : BOOL ;
     B13 : BOOL ;
     B14 : BOOL ;
     FABSPF : BOOL ;	//FABRICATION SANS PIECE AU FILM
     SPE : BOOL ;	//UNIT ESPECIAL
     B1 : BOOL ;
     B2 : BOOL ;
     B3 : BOOL ;
     B4 : BOOL ;
     B5 : BOOL ;
     B6 : BOOL ;
     B7 : BOOL ;
    END_STRUCT ;
    SPARE : ARRAY  [1 .. 4 ] OF INT ;
   END_STRUCT ;
   C0 : STRUCT 	//PART WORD C0
    MP : STRUCT 	//PART MEMORY / MOT PIECE
     MPP : BOOL ;	//PRESENT PART MEMORY / MEMOIRE PIECE PRESENTE
     MPAT : BOOL ;	//PART WITH WORK MEMORY / MEMOIRE PIECE A TRAVAILLER
     MPST : BOOL ;	//PART WITHOUT WORK MEMORY / MEMOIRE PIECE SANS TRAVAIL
     MPAM : BOOL ;	//PART MEMORY TO MATCH / MEMOIRE PIECE A MARIER
     MPAE : BOOL ;	//PART MEMORY TO EVACUATE / MEMOIRE PIECE A EVACUER
     MPP1 : BOOL ;	//INTERMEDIATE PRESENT PART MEMORY / MEMOIRE PIECE PRESENTE INTERMEDIAIRE
     MPP2 : BOOL ;	//INTERMEDIATE PRESENT PART MEMORY / MEMOIRE PIECE PRESENTE INTERMEDIAIRE
     MPP3 : BOOL ;	//INTERMEDIATE PRESENT PART MEMORY / MEMOIRE PIECE PRESENTE INTERMEDIAIRE
     MPP4 : BOOL ;	//INTERMEDIATE PRESENT PART MEMORY / MEMOIRE PIECE PRESENTE INTERMEDIAIRE
     MPP5 : BOOL ;	//INTERMEDIATE PRESENT PART MEMORY / MEMOIRE PIECE PRESENTE INTERMEDIAIRE
     MPP6 : BOOL ;	//INTERMEDIATE PRESENT PART MEMORY / MEMOIRE PIECE PRESENTE INTERMEDIAIRE
     MPP7 : BOOL ;	//INTERMEDIATE PRESENT PART MEMORY / MEMOIRE PIECE PRESENTE INTERMEDIAIRE
     MPP8 : BOOL ;	//INTERMEDIATE PRESENT PART MEMORY / MEMOIRE PIECE PRESENTE INTERMEDIAIRE
     MPT : BOOL ;	//PART COMPLETE MEMORY / MEMOIRE PIECE TRAVAILLE
     MPLNOK : BOOL ;	//LAUCHING PART MEMORY NOK / MEMOIRE LANCEMENT PIECE NON OK
     MPLNOR : BOOL ;	//LAUCHING PART MEMORY OK / MEMOIRE LANCEMENT PIECE OK
    END_STRUCT ;
    MS : STRUCT 	//SUPPORT WORD / MOT SUPPORT
     MSP : BOOL ;	//SUPPORT PRESENCE MEMORY / MEMOIRE SUPPORT PRESENT
     MSAE : BOOL ;	//SUPPORT TO EVACUATE MEMORY / MEMOIRE SUPPORT A EVACUER
     MSEBD : BOOL ;	//WRITING DATABASE SUPPORT MEMORY / MEMOIRE SUPPORT ECRITURE BASE DE DONNEE
     MSMBD : BOOL ;	//MODIFICATION DATABASE SUPPORT MEMORY / MEMOIRE SUPPORT MODIF BASE DE DONNEE
     MSLBD : BOOL ;	//READING DATABASE SUPPORT MEMORY / MEMOIRE SUPPORT LECTURE BASE DE DONNEE
     MSAP : BOOL ;	//PASSAGE AUTHORIZATION SUPPORT MEMORY / MEMOIRE SUPPORT AUTORISATION DE PASSAGE
     MRCPF : BOOL ;	//PART TO DO PROCESS CODE SEARCH MEMORY / MEMOIRE RECH CODES PROCESS A FAIRE
     MRCPS : BOOL ;	//NEXT PART PROCESS CODE SEARCH MEMORY / MEMOIRE RECH CODES PROCESS SUIVANT
     MSLRFID : BOOL ;	//READING RFID SUPPORT MEMORY / MEMOIRE SUPPORT LECTURE RFID
     MSERFID : BOOL ;	//WRITING RFID SUPPORT MEMORY / MEMOIRE SUPPORT ECRITURE RFID
     RES1 : BOOL ;	//SPARE / RESERVE
     RES2 : BOOL ;	//SPARE / RESERVE
     RES3 : BOOL ;	//SPARE / RESERVE
     RES4 : BOOL ;	//SPARE / RESERVE
     RES5 : BOOL ;	//SPARE / RESERVE
     RES6 : BOOL ;	//SPARE / RESERVE
    END_STRUCT ;
    NSUP : INT ;	//SUPPORT NUMBER / NUMERO DE SUPPORT
    NFILM : INT ;	//FILM NUMBER / NUMERO DE FILM
    NORDRE : INT ;	//ORDER NUMBER / NUMERO D ORDRE
    CDIV1 : INT ;	//FAMILIA / FAMILLE (CDIV1)
    CDIV2 : INT ;	//FASE / PHASE (CDIV2)
    CDIV3 : INT ;	//MODELO / MODELE (CDIV3)
    CDIV4 : INT ;	//TECHO (CDIV4)
    CDIV5 : INT ;	//VERSION (CDIV5)
    DESFI : INT ;	//FINAL DISPATCH / DESTINATION FINALE
    CSORT : INT ;	//CAUSE DE SORTIE
    DAT : STRUCT 	//DEFINITION / ATTENTE TRAVAIL
     B8 : BOOL ;	//PALETTE DE VIDAGE PERIMETRE (HORS SIPTOL)
     B9 : BOOL ;	//DEVERMINAGE PIECE / PALETTE (HORS SIPTOL)
     B10 : BOOL ;	//PALETTE DE MAP(HORS SIPTOL)
     B11 : BOOL ;	//PALETTE DE CHANGEMENT ELECTRODE BR (HORS SIPTOL)
     B12 : BOOL ;	//PALETTE DE CHANGEMENT ELECTRODE CS (HORS SIPTOL)
     B13 : BOOL ;	//DEVERMINAGE PIECE / PALETTE (AVEC SIPTOL)
     B14 : BOOL ;
     B15 : BOOL ;
     FABSPF : BOOL ;	//0 = AVEC TRAVAIL / 1 = SANS TRAVAIL (P1)
     B1 : BOOL ;
     B2 : BOOL ;	//0 = SUPPORT PLEIN / 1 = SUPPORT VIDE
     B3 : BOOL ;
     B4 : BOOL ;
     B5 : BOOL ;
     B6 : BOOL ;
     B7 : BOOL ;
    END_STRUCT ;
    CRAPI : STRUCT 	//PLC DISPATCHING REASON / CAUSE ROUTAGE API
     B8 : BOOL ;
     B9 : BOOL ;
     B10 : BOOL ;
     B11 : BOOL ;
     B12 : BOOL ;
     B13 : BOOL ;
     B14 : BOOL ;
     B15 : BOOL ;
     B0 : BOOL ;
     B1 : BOOL ;
     B2 : BOOL ;
     RARET : BOOL ;	//PIECE ANALYSE - RETOUCHE
     B4 : BOOL ;
     B5 : BOOL ;
     B6 : BOOL ;
     B7 : BOOL ;
    END_STRUCT ;
    MGEST : STRUCT 	//MOT DE GESTION RECALAGE
     MPFNOR : BOOL ;	//MEMOIRE PIECE FLUX NORMAL
     MPSTC : BOOL ;	//MEMOIRE PIECE A SORTIR TOUS CAS
     MPSOR : BOOL ;	//MEMOIRE PIECE A SORTIR (SORTIE SIPTOL BONNE)
     MPSSU : BOOL ;	//MEMOIRE PIECE A SORTIR (SUBTITUTION PIECE BONNE)
     MPSDI : BOOL ;	//MEMOIRE PIECE A SORTIR (DISCORDANCE)
     MPSSUL : BOOL ;	//MEMOIRE PIECE A SORTIR (SUBTITUTION PIECE LOUPEE)
     MPSL : BOOL ;	//MEMOIRE PIECE A SORTIR (SORTIE LOUPEE)
     MPSF99 : BOOL ;	//MEMOIRE PIECE A SORTIR (MAP FILM 99)
     MPETC : BOOL ;	//MEMOIRE PIECE A ENTRER TOUTS CAS
     MPEOR : BOOL ;	//MEMOIRE PIECE EN ENTREE (DEMANDE SIPTOL)
     MPESUB : BOOL ;	//MEMOIRE PIECE EN ENTREE (SUBTITUTION PIECE BONNE)
     MPEDI : BOOL ;	//MEMOIRE PIECE EN ENTREE (DISCORDANCE)
     MPESUL : BOOL ;	//MEMOIRE PIECE EN ENTREE (SUBTITUTION PIECE LOUPEE)
     MPOCV : BOOL ;	//MEMOIRE PIECE A SORTIR VEHICULE ANNULE + CROCHET VIDE
     MESUTC : BOOL ;	//MEMOIRE EN ENTREE SUBSTITUTION TOUS CAS (PIECE BONNE OU MAUVAISE)
     MSSUTC : BOOL ;	//MEMOIRE SORTIE SUBSTITUTION TOUS CAS (PIECE BONNE OU MAUVAISE)
    END_STRUCT ;
    TVEH : STRUCT 	//TYPO DE VEHICULO
     B8 : BOOL ;
     B9 : BOOL ;
     B10 : BOOL ;
     B11 : BOOL ;
     B12 : BOOL ;
     B13 : BOOL ;
     B14 : BOOL ;
     FABSPF : BOOL ;	//FABRICATION SANS PIECE AU FILM
     SPE : BOOL ;	//UNIT ESPECIAL
     B1 : BOOL ;
     B2 : BOOL ;
     B3 : BOOL ;
     B4 : BOOL ;
     B5 : BOOL ;
     B6 : BOOL ;
     B7 : BOOL ;
    END_STRUCT ;
    SPARE : ARRAY  [1 .. 4 ] OF INT ;	//SPARE
   END_STRUCT ;
   C0_TT : STRUCT 	//WORK TABLE C0
    MFT : STRUCT 	//END OF WORK MEMORY
     MFT1 : BOOL ;	//END OF WORK MEMORY 1 - SPARE
     MFT2 : BOOL ;	//END OF WORK MEMORY 2 - SPARE
     MFT3 : BOOL ;	//END OF WORK MEMORY 3 - SPARE
     MFT4 : BOOL ;	//END OF WORK MEMORY 4 - SPARE
     MFT5 : BOOL ;	//END OF WORK MEMORY 5 - SPARE
     MFT6 : BOOL ;	//END OF WORK MEMORY 6 - SPARE
     MFT7 : BOOL ;	//END OF WORK MEMORY 7 - SPARE
     MFT8 : BOOL ;	//END OF WORK MEMORY 8 - SPARE
     MFT9 : BOOL ;	//END OF WORK MEMORY 9 - SPARE
     MFT10 : BOOL ;	//END OF WORK MEMORY 10 - SPARE
     MFT11 : BOOL ;	//END OF WORK MEMORY 11 - SPARE
     MFT12 : BOOL ;	//END OF WORK MEMORY 12 - SPARE
     MFT13 : BOOL ;	//END OF WORK MEMORY 13 - SPARE
     MFT14 : BOOL ;	//END OF WORK MEMORY 14 - SPARE
     MFT15 : BOOL ;	//END OF WORK MEMORY 15 - SPARE
     MFT16 : BOOL ;	//END OF WORK MEMORY 16 - SPARE
    END_STRUCT ;
    C1 : STRUCT 	//END OF WORK MEMORY C1
     MFT1 : BOOL ;	//END OF WORK MEMORY 1 - SPARE
     MFT2 : BOOL ;	//END OF WORK MEMORY 2 - SPARE
     MFT3 : BOOL ;	//END OF WORK MEMORY 3 - SPARE
     MFT4 : BOOL ;	//END OF WORK MEMORY 4 - SPARE
     MFT5 : BOOL ;	//END OF WORK MEMORY 5 - SPARE
     MFT6 : BOOL ;	//END OF WORK MEMORY 6 - SPARE
     MFT7 : BOOL ;	//END OF WORK MEMORY 7 - SPARE
     MFT8 : BOOL ;	//END OF WORK MEMORY 8 - SPARE
    END_STRUCT ;
    C2 : STRUCT 	//END OF WORK MEMORY C2
     MFT1 : BOOL ;	//END OF WORK MEMORY 1 - SPARE
     MFT2 : BOOL ;	//END OF WORK MEMORY 2 - SPARE
     MFT3 : BOOL ;	//END OF WORK MEMORY 3 - SPARE
     MFT4 : BOOL ;	//END OF WORK MEMORY 4 - SPARE
     MFT5 : BOOL ;	//END OF WORK MEMORY 5 - SPARE
     MFT6 : BOOL ;	//END OF WORK MEMORY 6 - SPARE
     MFT7 : BOOL ;	//END OF WORK MEMORY 7 - SPARE
     MFT8 : BOOL ;	//END OF WORK MEMORY 8 - SPARE
    END_STRUCT ;
    SPARE : ARRAY  [1 .. 17 ] OF INT ;	//SPARE
   END_STRUCT ;
   D0 : STRUCT 	//PART WORD D0
    MP : STRUCT 	//PART MEMORY / MOT PIECE
     MPP : BOOL ;	//PRESENT PART MEMORY / MEMOIRE PIECE PRESENTE
     MPAT : BOOL ;	//PART WITH WORK MEMORY / MEMOIRE PIECE A TRAVAILLER
     MPST : BOOL ;	//PART WITHOUT WORK MEMORY / MEMOIRE PIECE SANS TRAVAIL
     MPAM : BOOL ;	//PART MEMORY TO MATCH / MEMOIRE PIECE A MARIER
     MPAE : BOOL ;	//PART MEMORY TO EVACUATE / MEMOIRE PIECE A EVACUER
     MPP1 : BOOL ;	//INTERMEDIATE PRESENT PART MEMORY / MEMOIRE PIECE PRESENTE INTERMEDIAIRE
     MPP2 : BOOL ;	//INTERMEDIATE PRESENT PART MEMORY / MEMOIRE PIECE PRESENTE INTERMEDIAIRE
     MPP3 : BOOL ;	//INTERMEDIATE PRESENT PART MEMORY / MEMOIRE PIECE PRESENTE INTERMEDIAIRE
     MPP4 : BOOL ;	//INTERMEDIATE PRESENT PART MEMORY / MEMOIRE PIECE PRESENTE INTERMEDIAIRE
     MPP5 : BOOL ;	//INTERMEDIATE PRESENT PART MEMORY / MEMOIRE PIECE PRESENTE INTERMEDIAIRE
     MPP6 : BOOL ;	//INTERMEDIATE PRESENT PART MEMORY / MEMOIRE PIECE PRESENTE INTERMEDIAIRE
     MPP7 : BOOL ;	//INTERMEDIATE PRESENT PART MEMORY / MEMOIRE PIECE PRESENTE INTERMEDIAIRE
     MPP8 : BOOL ;	//INTERMEDIATE PRESENT PART MEMORY / MEMOIRE PIECE PRESENTE INTERMEDIAIRE
     MPT : BOOL ;	//PART COMPLETE MEMORY / MEMOIRE PIECE TRAVAILLE
     MPLNOK : BOOL ;	//LAUCHING PART MEMORY NOK / MEMOIRE LANCEMENT PIECE NON OK
     MPLNOR : BOOL ;	//LAUCHING PART MEMORY OK / MEMOIRE LANCEMENT PIECE OK
    END_STRUCT ;
    MS : STRUCT 	//SUPPORT WORD / MOT SUPPORT
     MSP : BOOL ;	//SUPPORT PRESENCE MEMORY / MEMOIRE SUPPORT PRESENT
     MSAE : BOOL ;	//SUPPORT TO EVACUATE MEMORY / MEMOIRE SUPPORT A EVACUER
     MSEBD : BOOL ;	//WRITING DATABASE SUPPORT MEMORY / MEMOIRE SUPPORT ECRITURE BASE DE DONNEE
     MSMBD : BOOL ;	//MODIFICATION DATABASE SUPPORT MEMORY / MEMOIRE SUPPORT MODIF BASE DE DONNEE
     MSLBD : BOOL ;	//READING DATABASE SUPPORT MEMORY / MEMOIRE SUPPORT LECTURE BASE DE DONNEE
     MSAP : BOOL ;	//PASSAGE AUTHORIZATION SUPPORT MEMORY / MEMOIRE SUPPORT AUTORISATION DE PASSAGE
     MRCPF : BOOL ;	//PART TO DO PROCESS CODE SEARCH MEMORY / MEMOIRE RECH CODES PROCESS A FAIRE
     MRCPS : BOOL ;	//NEXT PART PROCESS CODE SEARCH MEMORY / MEMOIRE RECH CODES PROCESS SUIVANT
     MSLRFID : BOOL ;	//READING RFID SUPPORT MEMORY / MEMOIRE SUPPORT LECTURE RFID
     MSERFID : BOOL ;	//WRITING RFID SUPPORT MEMORY / MEMOIRE SUPPORT ECRITURE RFID
     RES1 : BOOL ;	//SPARE / RESERVE
     RES2 : BOOL ;	//SPARE / RESERVE
     RES3 : BOOL ;	//SPARE / RESERVE
     RES4 : BOOL ;	//SPARE / RESERVE
     RES5 : BOOL ;	//SPARE / RESERVE
     RES6 : BOOL ;	//SPARE / RESERVE
    END_STRUCT ;
    NSUP : INT ;	//SUPPORT NUMBER / NUMERO DE SUPPORT
    NFILM : INT ;	//FILM NUMBER / NUMERO DE FILM
    NORDRE : INT ;	//ORDER NUMBER / NUMERO D ORDRE
    CDIV1 : INT ;	//FAMILIA / FAMILLE (CDIV1)
    CDIV2 : INT ;	//FASE / PHASE (CDIV2)
    CDIV3 : INT ;	//MODELO / MODELE (CDIV3)
    CDIV4 : INT ;	//TECHO (CDIV4)
    CDIV5 : INT ;	//VERSION (CDIV5)
    DESFI : INT ;	//FINAL DISPATCH / DESTINATION FINALE
    CSORT : INT ;	//CAUSE DE SORTIE
    DAT : STRUCT 	//DEFINITION / ATTENTE TRAVAIL
     B8 : BOOL ;	//PALETTE DE VIDAGE PERIMETRE (HORS SIPTOL)
     B9 : BOOL ;	//DEVERMINAGE PIECE / PALETTE (HORS SIPTOL)
     B10 : BOOL ;	//PALETTE DE MAP(HORS SIPTOL)
     B11 : BOOL ;	//PALETTE DE CHANGEMENT ELECTRODE BR (HORS SIPTOL)
     B12 : BOOL ;	//PALETTE DE CHANGEMENT ELECTRODE CS (HORS SIPTOL)
     B13 : BOOL ;	//DEVERMINAGE PIECE / PALETTE (AVEC SIPTOL)
     B14 : BOOL ;
     B15 : BOOL ;
     FABSPF : BOOL ;	//0 = AVEC TRAVAIL / 1 = SANS TRAVAIL (P1)
     B1 : BOOL ;
     B2 : BOOL ;	//0 = SUPPORT PLEIN / 1 = SUPPORT VIDE
     B3 : BOOL ;
     B4 : BOOL ;
     B5 : BOOL ;
     B6 : BOOL ;
     B7 : BOOL ;
    END_STRUCT ;
    CRAPI : STRUCT 	//PLC DISPATCHING REASON / CAUSE ROUTAGE API
     B8 : BOOL ;
     B9 : BOOL ;
     B10 : BOOL ;
     B11 : BOOL ;
     B12 : BOOL ;
     B13 : BOOL ;
     B14 : BOOL ;
     B15 : BOOL ;
     B0 : BOOL ;
     B1 : BOOL ;
     B2 : BOOL ;
     RARET : BOOL ;	//PIECE ANALYSE - RETOUCHE
     B4 : BOOL ;
     B5 : BOOL ;
     B6 : BOOL ;
     B7 : BOOL ;
    END_STRUCT ;
    MGEST : STRUCT 	//MOT DE GESTION RECALAGE
     MPFNOR : BOOL ;	//MEMOIRE PIECE FLUX NORMAL
     MPSTC : BOOL ;	//MEMOIRE PIECE A SORTIR TOUS CAS
     MPSOR : BOOL ;	//MEMOIRE PIECE A SORTIR (SORTIE SIPTOL BONNE)
     MPSSU : BOOL ;	//MEMOIRE PIECE A SORTIR (SUBTITUTION PIECE BONNE)
     MPSDI : BOOL ;	//MEMOIRE PIECE A SORTIR (DISCORDANCE)
     MPSSUL : BOOL ;	//MEMOIRE PIECE A SORTIR (SUBTITUTION PIECE LOUPEE)
     MPSL : BOOL ;	//MEMOIRE PIECE A SORTIR (SORTIE LOUPEE)
     MPSF99 : BOOL ;	//MEMOIRE PIECE A SORTIR (MAP FILM 99)
     MPETC : BOOL ;	//MEMOIRE PIECE A ENTRER TOUTS CAS
     MPEOR : BOOL ;	//MEMOIRE PIECE EN ENTREE (DEMANDE SIPTOL)
     MPESUB : BOOL ;	//MEMOIRE PIECE EN ENTREE (SUBTITUTION PIECE BONNE)
     MPEDI : BOOL ;	//MEMOIRE PIECE EN ENTREE (DISCORDANCE)
     MPESUL : BOOL ;	//MEMOIRE PIECE EN ENTREE (SUBTITUTION PIECE LOUPEE)
     MPOCV : BOOL ;	//MEMOIRE PIECE A SORTIR VEHICULE ANNULE + CROCHET VIDE
     MESUTC : BOOL ;	//MEMOIRE EN ENTREE SUBSTITUTION TOUS CAS (PIECE BONNE OU MAUVAISE)
     MSSUTC : BOOL ;	//MEMOIRE SORTIE SUBSTITUTION TOUS CAS (PIECE BONNE OU MAUVAISE)
    END_STRUCT ;
    TVEH : STRUCT 	//TYPO DE VEHICULO
     B8 : BOOL ;
     B9 : BOOL ;
     B10 : BOOL ;
     B11 : BOOL ;
     B12 : BOOL ;
     B13 : BOOL ;
     B14 : BOOL ;
     FABSPF : BOOL ;	//FABRICATION SANS PIECE AU FILM
     SPE : BOOL ;	//UNIT ESPECIAL
     B1 : BOOL ;
     B2 : BOOL ;
     B3 : BOOL ;
     B4 : BOOL ;
     B5 : BOOL ;
     B6 : BOOL ;
     B7 : BOOL ;
    END_STRUCT ;
    SPARE : ARRAY  [1 .. 4 ] OF INT ;	//SPARE
   END_STRUCT ;
   D0_TT : STRUCT 	//WORK TABLE D0
    MFT : STRUCT 	//END OF WORK MEMORY
     MFT1 : BOOL ;	//END OF WORK MEMORY 1 - SPARE
     MFT2 : BOOL ;	//END OF WORK MEMORY 2 - SPARE
     MFT3 : BOOL ;	//END OF WORK MEMORY 3 - SPARE
     MFT4 : BOOL ;	//END OF WORK MEMORY 4 - SPARE
     MFT5 : BOOL ;	//END OF WORK MEMORY 5 - SPARE
     MFT6 : BOOL ;	//END OF WORK MEMORY 6 - SPARE
     MFT7 : BOOL ;	//END OF WORK MEMORY 7 - SPARE
     MFT8 : BOOL ;	//END OF WORK MEMORY 8 - SPARE
     MFT9 : BOOL ;	//END OF WORK MEMORY 9 - SPARE
     MFT10 : BOOL ;	//END OF WORK MEMORY 10 - SPARE
     MFT11 : BOOL ;	//END OF WORK MEMORY 11 - SPARE
     MFT12 : BOOL ;	//END OF WORK MEMORY 12 - SPARE
     MFT13 : BOOL ;	//END OF WORK MEMORY 13 - SPARE
     MFT14 : BOOL ;	//END OF WORK MEMORY 14 - SPARE
     MFT15 : BOOL ;	//END OF WORK MEMORY 15 - SPARE
     MFT16 : BOOL ;	//END OF WORK MEMORY 16 - SPARE
    END_STRUCT ;
    D1 : STRUCT 	//END OF WORK MEMORY D1
     MFT1 : BOOL ;	//END OF WORK MEMORY 1 - SPARE
     MFT2 : BOOL ;	//END OF WORK MEMORY 2 - SPARE
     MFT3 : BOOL ;	//END OF WORK MEMORY 3 - SPARE
     MFT4 : BOOL ;	//END OF WORK MEMORY 4 - SPARE
     MFT5 : BOOL ;	//END OF WORK MEMORY 5 - SPARE
     MFT6 : BOOL ;	//END OF WORK MEMORY 6 - SPARE
     MFT7 : BOOL ;	//END OF WORK MEMORY 7 - SPARE
     MFT8 : BOOL ;	//END OF WORK MEMORY 8 - SPARE
    END_STRUCT ;
    D2 : STRUCT 	//END OF WORK MEMORY D2
     MFT1 : BOOL ;	//END OF WORK MEMORY 1 - SPARE
     MFT2 : BOOL ;	//END OF WORK MEMORY 2 - SPARE
     MFT3 : BOOL ;	//END OF WORK MEMORY 3 - SPARE
     MFT4 : BOOL ;	//END OF WORK MEMORY 4 - SPARE
     MFT5 : BOOL ;	//END OF WORK MEMORY 5 - SPARE
     MFT6 : BOOL ;	//END OF WORK MEMORY 6 - SPARE
     MFT7 : BOOL ;	//END OF WORK MEMORY 7 - SPARE
     MFT8 : BOOL ;	//END OF WORK MEMORY 8 - SPARE
    END_STRUCT ;
    SPARE : ARRAY  [1 .. 17 ] OF INT ;	//SPARE
   END_STRUCT ;
   D0_GUINCHE : STRUCT 	//PART WORD D0 GUINCHE
    MP : STRUCT 	//PART MEMORY / MOT PIECE
     MPP : BOOL ;	//PRESENT PART MEMORY / MEMOIRE PIECE PRESENTE
     MPAT : BOOL ;	//PART WITH WORK MEMORY / MEMOIRE PIECE A TRAVAILLER
     MPST : BOOL ;	//PART WITHOUT WORK MEMORY / MEMOIRE PIECE SANS TRAVAIL
     MPAM : BOOL ;	//PART MEMORY TO MATCH / MEMOIRE PIECE A MARIER
     MPAE : BOOL ;	//PART MEMORY TO EVACUATE / MEMOIRE PIECE A EVACUER
     MPP1 : BOOL ;	//INTERMEDIATE PRESENT PART MEMORY / MEMOIRE PIECE PRESENTE INTERMEDIAIRE
     MPP2 : BOOL ;	//INTERMEDIATE PRESENT PART MEMORY / MEMOIRE PIECE PRESENTE INTERMEDIAIRE
     MPP3 : BOOL ;	//INTERMEDIATE PRESENT PART MEMORY / MEMOIRE PIECE PRESENTE INTERMEDIAIRE
     MPP4 : BOOL ;	//INTERMEDIATE PRESENT PART MEMORY / MEMOIRE PIECE PRESENTE INTERMEDIAIRE
     MPP5 : BOOL ;	//INTERMEDIATE PRESENT PART MEMORY / MEMOIRE PIECE PRESENTE INTERMEDIAIRE
     MPP6 : BOOL ;	//INTERMEDIATE PRESENT PART MEMORY / MEMOIRE PIECE PRESENTE INTERMEDIAIRE
     MPP7 : BOOL ;	//INTERMEDIATE PRESENT PART MEMORY / MEMOIRE PIECE PRESENTE INTERMEDIAIRE
     MPP8 : BOOL ;	//INTERMEDIATE PRESENT PART MEMORY / MEMOIRE PIECE PRESENTE INTERMEDIAIRE
     MPT : BOOL ;	//PART COMPLETE MEMORY / MEMOIRE PIECE TRAVAILLE
     MPLNOK : BOOL ;	//LAUCHING PART MEMORY NOK / MEMOIRE LANCEMENT PIECE NON OK
     MPLNOR : BOOL ;	//LAUCHING PART MEMORY OK / MEMOIRE LANCEMENT PIECE OK
    END_STRUCT ;
    MS : STRUCT 	//SUPPORT WORD / MOT SUPPORT
     MSP : BOOL ;	//SUPPORT PRESENCE MEMORY / MEMOIRE SUPPORT PRESENT
     MSAE : BOOL ;	//SUPPORT TO EVACUATE MEMORY / MEMOIRE SUPPORT A EVACUER
     MSEBD : BOOL ;	//WRITING DATABASE SUPPORT MEMORY / MEMOIRE SUPPORT ECRITURE BASE DE DONNEE
     MSMBD : BOOL ;	//MODIFICATION DATABASE SUPPORT MEMORY / MEMOIRE SUPPORT MODIF BASE DE DONNEE
     MSLBD : BOOL ;	//READING DATABASE SUPPORT MEMORY / MEMOIRE SUPPORT LECTURE BASE DE DONNEE
     MSAP : BOOL ;	//PASSAGE AUTHORIZATION SUPPORT MEMORY / MEMOIRE SUPPORT AUTORISATION DE PASSAGE
     MRCPF : BOOL ;	//PART TO DO PROCESS CODE SEARCH MEMORY / MEMOIRE RECH CODES PROCESS A FAIRE
     MRCPS : BOOL ;	//NEXT PART PROCESS CODE SEARCH MEMORY / MEMOIRE RECH CODES PROCESS SUIVANT
     MSLRFID : BOOL ;	//READING RFID SUPPORT MEMORY / MEMOIRE SUPPORT LECTURE RFID
     MSERFID : BOOL ;	//WRITING RFID SUPPORT MEMORY / MEMOIRE SUPPORT ECRITURE RFID
     RES1 : BOOL ;	//SPARE / RESERVE
     RES2 : BOOL ;	//SPARE / RESERVE
     RES3 : BOOL ;	//SPARE / RESERVE
     RES4 : BOOL ;	//SPARE / RESERVE
     RES5 : BOOL ;	//SPARE / RESERVE
     RES6 : BOOL ;	//SPARE / RESERVE
    END_STRUCT ;
    NSUP : INT ;	//SUPPORT NUMBER / NUMERO DE SUPPORT
    NFILM : INT ;	//FILM NUMBER / NUMERO DE FILM
    NORDRE : INT ;	//ORDER NUMBER / NUMERO D ORDRE
    CDIV1 : INT ;	//FAMILIA / FAMILLE (CDIV1)
    CDIV2 : INT ;	//FASE / PHASE (CDIV2)
    CDIV3 : INT ;	//MODELO / MODELE (CDIV3)
    CDIV4 : INT ;	//TECHO (CDIV4)
    CDIV5 : INT ;	//VERSION (CDIV5)
    DESFI : INT ;	//FINAL DISPATCH / DESTINATION FINALE
    CSORT : INT ;	//CAUSE DE SORTIE
    DAT : STRUCT 	//DEFINITION / ATTENTE TRAVAIL
     B8 : BOOL ;	//PALETTE DE VIDAGE PERIMETRE (HORS SIPTOL)
     B9 : BOOL ;	//DEVERMINAGE PIECE / PALETTE (HORS SIPTOL)
     B10 : BOOL ;	//PALETTE DE MAP(HORS SIPTOL)
     B11 : BOOL ;	//PALETTE DE CHANGEMENT ELECTRODE BR (HORS SIPTOL)
     B12 : BOOL ;	//PALETTE DE CHANGEMENT ELECTRODE CS (HORS SIPTOL)
     B13 : BOOL ;	//DEVERMINAGE PIECE / PALETTE (AVEC SIPTOL)
     B14 : BOOL ;
     B15 : BOOL ;
     FABSPF : BOOL ;	//0 = AVEC TRAVAIL / 1 = SANS TRAVAIL (P1)
     B1 : BOOL ;
     B2 : BOOL ;	//0 = SUPPORT PLEIN / 1 = SUPPORT VIDE
     B3 : BOOL ;
     B4 : BOOL ;
     B5 : BOOL ;
     B6 : BOOL ;
     B7 : BOOL ;
    END_STRUCT ;
    CRAPI : STRUCT 	//PLC DISPATCHING REASON / CAUSE ROUTAGE API
     B8 : BOOL ;
     B9 : BOOL ;
     B10 : BOOL ;
     B11 : BOOL ;
     B12 : BOOL ;
     B13 : BOOL ;
     B14 : BOOL ;
     B15 : BOOL ;
     B0 : BOOL ;
     B1 : BOOL ;
     B2 : BOOL ;
     RARET : BOOL ;	//PIECE ANALYSE - RETOUCHE
     B4 : BOOL ;
     B5 : BOOL ;
     B6 : BOOL ;
     B7 : BOOL ;
    END_STRUCT ;
    MGEST : STRUCT 	//MOT DE GESTION RECALAGE
     MPFNOR : BOOL ;	//MEMOIRE PIECE FLUX NORMAL
     MPSTC : BOOL ;	//MEMOIRE PIECE A SORTIR TOUS CAS
     MPSOR : BOOL ;	//MEMOIRE PIECE A SORTIR (SORTIE SIPTOL BONNE)
     MPSSU : BOOL ;	//MEMOIRE PIECE A SORTIR (SUBTITUTION PIECE BONNE)
     MPSDI : BOOL ;	//MEMOIRE PIECE A SORTIR (DISCORDANCE)
     MPSSUL : BOOL ;	//MEMOIRE PIECE A SORTIR (SUBTITUTION PIECE LOUPEE)
     MPSL : BOOL ;	//MEMOIRE PIECE A SORTIR (SORTIE LOUPEE)
     MPSF99 : BOOL ;	//MEMOIRE PIECE A SORTIR (MAP FILM 99)
     MPETC : BOOL ;	//MEMOIRE PIECE A ENTRER TOUTS CAS
     MPEOR : BOOL ;	//MEMOIRE PIECE EN ENTREE (DEMANDE SIPTOL)
     MPESUB : BOOL ;	//MEMOIRE PIECE EN ENTREE (SUBTITUTION PIECE BONNE)
     MPEDI : BOOL ;	//MEMOIRE PIECE EN ENTREE (DISCORDANCE)
     MPESUL : BOOL ;	//MEMOIRE PIECE EN ENTREE (SUBTITUTION PIECE LOUPEE)
     MPOCV : BOOL ;	//MEMOIRE PIECE A SORTIR VEHICULE ANNULE + CROCHET VIDE
     MESUTC : BOOL ;	//MEMOIRE EN ENTREE SUBSTITUTION TOUS CAS (PIECE BONNE OU MAUVAISE)
     MSSUTC : BOOL ;	//MEMOIRE SORTIE SUBSTITUTION TOUS CAS (PIECE BONNE OU MAUVAISE)
    END_STRUCT ;
    TVEH : STRUCT 	//TYPO DE VEHICULO
     B8 : BOOL ;
     B9 : BOOL ;
     B10 : BOOL ;
     B11 : BOOL ;
     B12 : BOOL ;
     B13 : BOOL ;
     B14 : BOOL ;
     FABSPF : BOOL ;	//FABRICATION SANS PIECE AU FILM
     SPE : BOOL ;	//UNIT ESPECIAL
     B1 : BOOL ;
     B2 : BOOL ;
     B3 : BOOL ;
     B4 : BOOL ;
     B5 : BOOL ;
     B6 : BOOL ;
     B7 : BOOL ;
    END_STRUCT ;
    SPARE : ARRAY  [1 .. 4 ] OF INT ;
   END_STRUCT ;
   LD : STRUCT 	//PART WORD D0
    MP : STRUCT 	//PART MEMORY / MOT PIECE
     MPP : BOOL ;	//PRESENT PART MEMORY / MEMOIRE PIECE PRESENTE
     MPAT : BOOL ;	//PART WITH WORK MEMORY / MEMOIRE PIECE A TRAVAILLER
     MPST : BOOL ;	//PART WITHOUT WORK MEMORY / MEMOIRE PIECE SANS TRAVAIL
     MPAM : BOOL ;	//PART MEMORY TO MATCH / MEMOIRE PIECE A MARIER
     MPAE : BOOL ;	//PART MEMORY TO EVACUATE / MEMOIRE PIECE A EVACUER
     MPP1 : BOOL ;	//INTERMEDIATE PRESENT PART MEMORY / MEMOIRE PIECE PRESENTE INTERMEDIAIRE
     MPP2 : BOOL ;	//INTERMEDIATE PRESENT PART MEMORY / MEMOIRE PIECE PRESENTE INTERMEDIAIRE
     MPP3 : BOOL ;	//INTERMEDIATE PRESENT PART MEMORY / MEMOIRE PIECE PRESENTE INTERMEDIAIRE
     MPP4 : BOOL ;	//INTERMEDIATE PRESENT PART MEMORY / MEMOIRE PIECE PRESENTE INTERMEDIAIRE
     MPP5 : BOOL ;	//INTERMEDIATE PRESENT PART MEMORY / MEMOIRE PIECE PRESENTE INTERMEDIAIRE
     MPP6 : BOOL ;	//INTERMEDIATE PRESENT PART MEMORY / MEMOIRE PIECE PRESENTE INTERMEDIAIRE
     MPP7 : BOOL ;	//INTERMEDIATE PRESENT PART MEMORY / MEMOIRE PIECE PRESENTE INTERMEDIAIRE
     MPP8 : BOOL ;	//INTERMEDIATE PRESENT PART MEMORY / MEMOIRE PIECE PRESENTE INTERMEDIAIRE
     MPT : BOOL ;	//PART COMPLETE MEMORY / MEMOIRE PIECE TRAVAILLE
     MPLNOK : BOOL ;	//LAUCHING PART MEMORY NOK / MEMOIRE LANCEMENT PIECE NON OK
     MPLNOR : BOOL ;	//LAUCHING PART MEMORY OK / MEMOIRE LANCEMENT PIECE OK
    END_STRUCT ;
    MS : STRUCT 	//SUPPORT WORD / MOT SUPPORT
     MSP : BOOL ;	//SUPPORT PRESENCE MEMORY / MEMOIRE SUPPORT PRESENT
     MSAE : BOOL ;	//SUPPORT TO EVACUATE MEMORY / MEMOIRE SUPPORT A EVACUER
     MSEBD : BOOL ;	//WRITING DATABASE SUPPORT MEMORY / MEMOIRE SUPPORT ECRITURE BASE DE DONNEE
     MSMBD : BOOL ;	//MODIFICATION DATABASE SUPPORT MEMORY / MEMOIRE SUPPORT MODIF BASE DE DONNEE
     MSLBD : BOOL ;	//READING DATABASE SUPPORT MEMORY / MEMOIRE SUPPORT LECTURE BASE DE DONNEE
     MSAP : BOOL ;	//PASSAGE AUTHORIZATION SUPPORT MEMORY / MEMOIRE SUPPORT AUTORISATION DE PASSAGE
     MRCPF : BOOL ;	//PART TO DO PROCESS CODE SEARCH MEMORY / MEMOIRE RECH CODES PROCESS A FAIRE
     MRCPS : BOOL ;	//NEXT PART PROCESS CODE SEARCH MEMORY / MEMOIRE RECH CODES PROCESS SUIVANT
     MSLRFID : BOOL ;	//READING RFID SUPPORT MEMORY / MEMOIRE SUPPORT LECTURE RFID
     MSERFID : BOOL ;	//WRITING RFID SUPPORT MEMORY / MEMOIRE SUPPORT ECRITURE RFID
     RES1 : BOOL ;	//SPARE / RESERVE
     RES2 : BOOL ;	//SPARE / RESERVE
     RES3 : BOOL ;	//SPARE / RESERVE
     RES4 : BOOL ;	//SPARE / RESERVE
     RES5 : BOOL ;	//SPARE / RESERVE
     RES6 : BOOL ;	//SPARE / RESERVE
    END_STRUCT ;
    NSUP : INT ;	//SUPPORT NUMBER / NUMERO DE SUPPORT
    NFILM : INT ;	//FILM NUMBER / NUMERO DE FILM
    NORDRE : INT ;	//ORDER NUMBER / NUMERO D ORDRE
    CDIV1 : INT ;	//FAMILIA / FAMILLE (CDIV1)
    CDIV2 : INT ;	//FASE / PHASE (CDIV2)
    CDIV3 : INT ;	//MODELO / MODELE (CDIV3)
    CDIV4 : INT ;	//TECHO (CDIV4)
    CDIV5 : INT ;	//VERSION (CDIV5)
    DESFI : INT ;	//FINAL DISPATCH / DESTINATION FINALE
    CSORT : INT ;	//CAUSE DE SORTIE
    DAT : STRUCT 	//DEFINITION / ATTENTE TRAVAIL
     B8 : BOOL ;	//PALETTE DE VIDAGE PERIMETRE (HORS SIPTOL)
     B9 : BOOL ;	//DEVERMINAGE PIECE / PALETTE (HORS SIPTOL)
     B10 : BOOL ;	//PALETTE DE MAP(HORS SIPTOL)
     B11 : BOOL ;	//PALETTE DE CHANGEMENT ELECTRODE BR (HORS SIPTOL)
     B12 : BOOL ;	//PALETTE DE CHANGEMENT ELECTRODE CS (HORS SIPTOL)
     B13 : BOOL ;	//DEVERMINAGE PIECE / PALETTE (AVEC SIPTOL)
     B14 : BOOL ;
     B15 : BOOL ;
     FABSPF : BOOL ;	//0 = AVEC TRAVAIL / 1 = SANS TRAVAIL (P1)
     B1 : BOOL ;
     B2 : BOOL ;	//0 = SUPPORT PLEIN / 1 = SUPPORT VIDE
     B3 : BOOL ;
     B4 : BOOL ;
     B5 : BOOL ;
     B6 : BOOL ;
     B7 : BOOL ;
    END_STRUCT ;
    CRAPI : STRUCT 	//PLC DISPATCHING REASON / CAUSE ROUTAGE API
     B8 : BOOL ;
     B9 : BOOL ;
     B10 : BOOL ;
     B11 : BOOL ;
     B12 : BOOL ;
     B13 : BOOL ;
     B14 : BOOL ;
     B15 : BOOL ;
     B0 : BOOL ;
     B1 : BOOL ;
     B2 : BOOL ;
     RARET : BOOL ;	//PIECE ANALYSE - RETOUCHE
     B4 : BOOL ;
     B5 : BOOL ;
     B6 : BOOL ;
     B7 : BOOL ;
    END_STRUCT ;
    MGEST : STRUCT 	//MOT DE GESTION RECALAGE
     MPFNOR : BOOL ;	//MEMOIRE PIECE FLUX NORMAL
     MPSTC : BOOL ;	//MEMOIRE PIECE A SORTIR TOUS CAS
     MPSOR : BOOL ;	//MEMOIRE PIECE A SORTIR (SORTIE SIPTOL BONNE)
     MPSSU : BOOL ;	//MEMOIRE PIECE A SORTIR (SUBTITUTION PIECE BONNE)
     MPSDI : BOOL ;	//MEMOIRE PIECE A SORTIR (DISCORDANCE)
     MPSSUL : BOOL ;	//MEMOIRE PIECE A SORTIR (SUBTITUTION PIECE LOUPEE)
     MPSL : BOOL ;	//MEMOIRE PIECE A SORTIR (SORTIE LOUPEE)
     MPSF99 : BOOL ;	//MEMOIRE PIECE A SORTIR (MAP FILM 99)
     MPETC : BOOL ;	//MEMOIRE PIECE A ENTRER TOUTS CAS
     MPEOR : BOOL ;	//MEMOIRE PIECE EN ENTREE (DEMANDE SIPTOL)
     MPESUB : BOOL ;	//MEMOIRE PIECE EN ENTREE (SUBTITUTION PIECE BONNE)
     MPEDI : BOOL ;	//MEMOIRE PIECE EN ENTREE (DISCORDANCE)
     MPESUL : BOOL ;	//MEMOIRE PIECE EN ENTREE (SUBTITUTION PIECE LOUPEE)
     MPOCV : BOOL ;	//MEMOIRE PIECE A SORTIR VEHICULE ANNULE + CROCHET VIDE
     MESUTC : BOOL ;	//MEMOIRE EN ENTREE SUBSTITUTION TOUS CAS (PIECE BONNE OU MAUVAISE)
     MSSUTC : BOOL ;	//MEMOIRE SORTIE SUBSTITUTION TOUS CAS (PIECE BONNE OU MAUVAISE)
    END_STRUCT ;
    TVEH : STRUCT 	//TYPO DE VEHICULO
     B8 : BOOL ;
     B9 : BOOL ;
     B10 : BOOL ;
     B11 : BOOL ;
     B12 : BOOL ;
     B13 : BOOL ;
     B14 : BOOL ;
     FABSPF : BOOL ;	//FABRICATION SANS PIECE AU FILM
     SPE : BOOL ;	//UNIT ESPECIAL
     B1 : BOOL ;
     B2 : BOOL ;
     B3 : BOOL ;
     B4 : BOOL ;
     B5 : BOOL ;
     B6 : BOOL ;
     B7 : BOOL ;
    END_STRUCT ;
    SPARE : ARRAY  [1 .. 4 ] OF INT ;
   END_STRUCT ;
   LD_TT : STRUCT 	//WORK TABLE D0
    MFT : STRUCT 	//END OF WORK MEMORY
     MFT1 : BOOL ;	//END OF WORK MEMORY 1 - SPARE
     MFT2 : BOOL ;	//END OF WORK MEMORY 2 - SPARE
     MFT3 : BOOL ;	//END OF WORK MEMORY 3 - SPARE
     MFT4 : BOOL ;	//END OF WORK MEMORY 4 - SPARE
     MFT5 : BOOL ;	//END OF WORK MEMORY 5 - SPARE
     MFT6 : BOOL ;	//END OF WORK MEMORY 6 - SPARE
     MFT7 : BOOL ;	//END OF WORK MEMORY 7 - SPARE
     MFT8 : BOOL ;	//END OF WORK MEMORY 8 - SPARE
     MFT9 : BOOL ;	//END OF WORK MEMORY 9 - SPARE
     MFT10 : BOOL ;	//END OF WORK MEMORY 10 - SPARE
     MFT11 : BOOL ;	//END OF WORK MEMORY 11 - SPARE
     MFT12 : BOOL ;	//END OF WORK MEMORY 12 - SPARE
     MFT13 : BOOL ;	//END OF WORK MEMORY 13 - SPARE
     MFT14 : BOOL ;	//END OF WORK MEMORY 14 - SPARE
     MFT15 : BOOL ;	//END OF WORK MEMORY 15 - SPARE
     MFT16 : BOOL ;	//END OF WORK MEMORY 16 - SPARE
    END_STRUCT ;
    LD1 : STRUCT 	//END OF WORK MEMORY D1
     MFT1 : BOOL ;	//END OF WORK MEMORY 1 - SPARE
     MFT2 : BOOL ;	//END OF WORK MEMORY 2 - SPARE
     MFT3 : BOOL ;	//END OF WORK MEMORY 3 - SPARE
     MFT4 : BOOL ;	//END OF WORK MEMORY 4 - SPARE
     MFT5 : BOOL ;	//END OF WORK MEMORY 5 - SPARE
     MFT6 : BOOL ;	//END OF WORK MEMORY 6 - SPARE
     MFT7 : BOOL ;	//END OF WORK MEMORY 7 - SPARE
     MFT8 : BOOL ;	//END OF WORK MEMORY 8 - SPARE
    END_STRUCT ;
    LD2 : STRUCT 	//END OF WORK MEMORY D2
     MFT1 : BOOL ;	//END OF WORK MEMORY 1 - SPARE
     MFT2 : BOOL ;	//END OF WORK MEMORY 2 - SPARE
     MFT3 : BOOL ;	//END OF WORK MEMORY 3 - SPARE
     MFT4 : BOOL ;	//END OF WORK MEMORY 4 - SPARE
     MFT5 : BOOL ;	//END OF WORK MEMORY 5 - SPARE
     MFT6 : BOOL ;	//END OF WORK MEMORY 6 - SPARE
     MFT7 : BOOL ;	//END OF WORK MEMORY 7 - SPARE
     MFT8 : BOOL ;	//END OF WORK MEMORY 8 - SPARE
    END_STRUCT ;
    SPARE : ARRAY  [1 .. 17 ] OF INT ;
   END_STRUCT ;
   LG : STRUCT 	//PART WORD D0
    MP : STRUCT 	//PART MEMORY / MOT PIECE
     MPP : BOOL ;	//PRESENT PART MEMORY / MEMOIRE PIECE PRESENTE
     MPAT : BOOL ;	//PART WITH WORK MEMORY / MEMOIRE PIECE A TRAVAILLER
     MPST : BOOL ;	//PART WITHOUT WORK MEMORY / MEMOIRE PIECE SANS TRAVAIL
     MPAM : BOOL ;	//PART MEMORY TO MATCH / MEMOIRE PIECE A MARIER
     MPAE : BOOL ;	//PART MEMORY TO EVACUATE / MEMOIRE PIECE A EVACUER
     MPP1 : BOOL ;	//INTERMEDIATE PRESENT PART MEMORY / MEMOIRE PIECE PRESENTE INTERMEDIAIRE
     MPP2 : BOOL ;	//INTERMEDIATE PRESENT PART MEMORY / MEMOIRE PIECE PRESENTE INTERMEDIAIRE
     MPP3 : BOOL ;	//INTERMEDIATE PRESENT PART MEMORY / MEMOIRE PIECE PRESENTE INTERMEDIAIRE
     MPP4 : BOOL ;	//INTERMEDIATE PRESENT PART MEMORY / MEMOIRE PIECE PRESENTE INTERMEDIAIRE
     MPP5 : BOOL ;	//INTERMEDIATE PRESENT PART MEMORY / MEMOIRE PIECE PRESENTE INTERMEDIAIRE
     MPP6 : BOOL ;	//INTERMEDIATE PRESENT PART MEMORY / MEMOIRE PIECE PRESENTE INTERMEDIAIRE
     MPP7 : BOOL ;	//INTERMEDIATE PRESENT PART MEMORY / MEMOIRE PIECE PRESENTE INTERMEDIAIRE
     MPP8 : BOOL ;	//INTERMEDIATE PRESENT PART MEMORY / MEMOIRE PIECE PRESENTE INTERMEDIAIRE
     MPT : BOOL ;	//PART COMPLETE MEMORY / MEMOIRE PIECE TRAVAILLE
     MPLNOK : BOOL ;	//LAUCHING PART MEMORY NOK / MEMOIRE LANCEMENT PIECE NON OK
     MPLNOR : BOOL ;	//LAUCHING PART MEMORY OK / MEMOIRE LANCEMENT PIECE OK
    END_STRUCT ;
    MS : STRUCT 	//SUPPORT WORD / MOT SUPPORT
     MSP : BOOL ;	//SUPPORT PRESENCE MEMORY / MEMOIRE SUPPORT PRESENT
     MSAE : BOOL ;	//SUPPORT TO EVACUATE MEMORY / MEMOIRE SUPPORT A EVACUER
     MSEBD : BOOL ;	//WRITING DATABASE SUPPORT MEMORY / MEMOIRE SUPPORT ECRITURE BASE DE DONNEE
     MSMBD : BOOL ;	//MODIFICATION DATABASE SUPPORT MEMORY / MEMOIRE SUPPORT MODIF BASE DE DONNEE
     MSLBD : BOOL ;	//READING DATABASE SUPPORT MEMORY / MEMOIRE SUPPORT LECTURE BASE DE DONNEE
     MSAP : BOOL ;	//PASSAGE AUTHORIZATION SUPPORT MEMORY / MEMOIRE SUPPORT AUTORISATION DE PASSAGE
     MRCPF : BOOL ;	//PART TO DO PROCESS CODE SEARCH MEMORY / MEMOIRE RECH CODES PROCESS A FAIRE
     MRCPS : BOOL ;	//NEXT PART PROCESS CODE SEARCH MEMORY / MEMOIRE RECH CODES PROCESS SUIVANT
     MSLRFID : BOOL ;	//READING RFID SUPPORT MEMORY / MEMOIRE SUPPORT LECTURE RFID
     MSERFID : BOOL ;	//WRITING RFID SUPPORT MEMORY / MEMOIRE SUPPORT ECRITURE RFID
     RES1 : BOOL ;	//SPARE / RESERVE
     RES2 : BOOL ;	//SPARE / RESERVE
     RES3 : BOOL ;	//SPARE / RESERVE
     RES4 : BOOL ;	//SPARE / RESERVE
     RES5 : BOOL ;	//SPARE / RESERVE
     RES6 : BOOL ;	//SPARE / RESERVE
    END_STRUCT ;
    NSUP : INT ;	//SUPPORT NUMBER / NUMERO DE SUPPORT
    NFILM : INT ;	//FILM NUMBER / NUMERO DE FILM
    NORDRE : INT ;	//ORDER NUMBER / NUMERO D ORDRE
    CDIV1 : INT ;	//FAMILIA / FAMILLE (CDIV1)
    CDIV2 : INT ;	//FASE / PHASE (CDIV2)
    CDIV3 : INT ;	//MODELO / MODELE (CDIV3)
    CDIV4 : INT ;	//TECHO (CDIV4)
    CDIV5 : INT ;	//VERSION (CDIV5)
    DESFI : INT ;	//FINAL DISPATCH / DESTINATION FINALE
    CSORT : INT ;	//CAUSE DE SORTIE
    DAT : STRUCT 	//DEFINITION / ATTENTE TRAVAIL
     B8 : BOOL ;	//PALETTE DE VIDAGE PERIMETRE (HORS SIPTOL)
     B9 : BOOL ;	//DEVERMINAGE PIECE / PALETTE (HORS SIPTOL)
     B10 : BOOL ;	//PALETTE DE MAP(HORS SIPTOL)
     B11 : BOOL ;	//PALETTE DE CHANGEMENT ELECTRODE BR (HORS SIPTOL)
     B12 : BOOL ;	//PALETTE DE CHANGEMENT ELECTRODE CS (HORS SIPTOL)
     B13 : BOOL ;	//DEVERMINAGE PIECE / PALETTE (AVEC SIPTOL)
     B14 : BOOL ;
     B15 : BOOL ;
     FABSPF : BOOL ;	//0 = AVEC TRAVAIL / 1 = SANS TRAVAIL (P1)
     B1 : BOOL ;
     B2 : BOOL ;	//0 = SUPPORT PLEIN / 1 = SUPPORT VIDE
     B3 : BOOL ;
     B4 : BOOL ;
     B5 : BOOL ;
     B6 : BOOL ;
     B7 : BOOL ;
    END_STRUCT ;
    CRAPI : STRUCT 	//PLC DISPATCHING REASON / CAUSE ROUTAGE API
     B8 : BOOL ;
     B9 : BOOL ;
     B10 : BOOL ;
     B11 : BOOL ;
     B12 : BOOL ;
     B13 : BOOL ;
     B14 : BOOL ;
     B15 : BOOL ;
     B0 : BOOL ;
     B1 : BOOL ;
     B2 : BOOL ;
     RARET : BOOL ;	//PIECE ANALYSE - RETOUCHE
     B4 : BOOL ;
     B5 : BOOL ;
     B6 : BOOL ;
     B7 : BOOL ;
    END_STRUCT ;
    MGEST : STRUCT 	//MOT DE GESTION RECALAGE
     MPFNOR : BOOL ;	//MEMOIRE PIECE FLUX NORMAL
     MPSTC : BOOL ;	//MEMOIRE PIECE A SORTIR TOUS CAS
     MPSOR : BOOL ;	//MEMOIRE PIECE A SORTIR (SORTIE SIPTOL BONNE)
     MPSSU : BOOL ;	//MEMOIRE PIECE A SORTIR (SUBTITUTION PIECE BONNE)
     MPSDI : BOOL ;	//MEMOIRE PIECE A SORTIR (DISCORDANCE)
     MPSSUL : BOOL ;	//MEMOIRE PIECE A SORTIR (SUBTITUTION PIECE LOUPEE)
     MPSL : BOOL ;	//MEMOIRE PIECE A SORTIR (SORTIE LOUPEE)
     MPSF99 : BOOL ;	//MEMOIRE PIECE A SORTIR (MAP FILM 99)
     MPETC : BOOL ;	//MEMOIRE PIECE A ENTRER TOUTS CAS
     MPEOR : BOOL ;	//MEMOIRE PIECE EN ENTREE (DEMANDE SIPTOL)
     MPESUB : BOOL ;	//MEMOIRE PIECE EN ENTREE (SUBTITUTION PIECE BONNE)
     MPEDI : BOOL ;	//MEMOIRE PIECE EN ENTREE (DISCORDANCE)
     MPESUL : BOOL ;	//MEMOIRE PIECE EN ENTREE (SUBTITUTION PIECE LOUPEE)
     MPOCV : BOOL ;	//MEMOIRE PIECE A SORTIR VEHICULE ANNULE + CROCHET VIDE
     MESUTC : BOOL ;	//MEMOIRE EN ENTREE SUBSTITUTION TOUS CAS (PIECE BONNE OU MAUVAISE)
     MSSUTC : BOOL ;	//MEMOIRE SORTIE SUBSTITUTION TOUS CAS (PIECE BONNE OU MAUVAISE)
    END_STRUCT ;
    TVEH : STRUCT 	//TYPO DE VEHICULO
     B8 : BOOL ;
     B9 : BOOL ;
     B10 : BOOL ;
     B11 : BOOL ;
     B12 : BOOL ;
     B13 : BOOL ;
     B14 : BOOL ;
     FABSPF : BOOL ;	//FABRICATION SANS PIECE AU FILM
     SPE : BOOL ;	//UNIT ESPECIAL
     B1 : BOOL ;
     B2 : BOOL ;
     B3 : BOOL ;
     B4 : BOOL ;
     B5 : BOOL ;
     B6 : BOOL ;
     B7 : BOOL ;
    END_STRUCT ;
    SPARE : ARRAY  [1 .. 4 ] OF INT ;
   END_STRUCT ;
   LG_TT : STRUCT 	//WORK TABLE D0
    MFT : STRUCT 	//END OF WORK MEMORY
     MFT1 : BOOL ;	//END OF WORK MEMORY 1 - SPARE
     MFT2 : BOOL ;	//END OF WORK MEMORY 2 - SPARE
     MFT3 : BOOL ;	//END OF WORK MEMORY 3 - SPARE
     MFT4 : BOOL ;	//END OF WORK MEMORY 4 - SPARE
     MFT5 : BOOL ;	//END OF WORK MEMORY 5 - SPARE
     MFT6 : BOOL ;	//END OF WORK MEMORY 6 - SPARE
     MFT7 : BOOL ;	//END OF WORK MEMORY 7 - SPARE
     MFT8 : BOOL ;	//END OF WORK MEMORY 8 - SPARE
     MFT9 : BOOL ;	//END OF WORK MEMORY 9 - SPARE
     MFT10 : BOOL ;	//END OF WORK MEMORY 10 - SPARE
     MFT11 : BOOL ;	//END OF WORK MEMORY 11 - SPARE
     MFT12 : BOOL ;	//END OF WORK MEMORY 12 - SPARE
     MFT13 : BOOL ;	//END OF WORK MEMORY 13 - SPARE
     MFT14 : BOOL ;	//END OF WORK MEMORY 14 - SPARE
     MFT15 : BOOL ;	//END OF WORK MEMORY 15 - SPARE
     MFT16 : BOOL ;	//END OF WORK MEMORY 16 - SPARE
    END_STRUCT ;
    LG1 : STRUCT 	//END OF WORK MEMORY D1
     MFT1 : BOOL ;	//END OF WORK MEMORY 1 - SPARE
     MFT2 : BOOL ;	//END OF WORK MEMORY 2 - SPARE
     MFT3 : BOOL ;	//END OF WORK MEMORY 3 - SPARE
     MFT4 : BOOL ;	//END OF WORK MEMORY 4 - SPARE
     MFT5 : BOOL ;	//END OF WORK MEMORY 5 - SPARE
     MFT6 : BOOL ;	//END OF WORK MEMORY 6 - SPARE
     MFT7 : BOOL ;	//END OF WORK MEMORY 7 - SPARE
     MFT8 : BOOL ;	//END OF WORK MEMORY 8 - SPARE
    END_STRUCT ;
    LG2 : STRUCT 	//END OF WORK MEMORY D2
     MFT1 : BOOL ;	//END OF WORK MEMORY 1 - SPARE
     MFT2 : BOOL ;	//END OF WORK MEMORY 2 - SPARE
     MFT3 : BOOL ;	//END OF WORK MEMORY 3 - SPARE
     MFT4 : BOOL ;	//END OF WORK MEMORY 4 - SPARE
     MFT5 : BOOL ;	//END OF WORK MEMORY 5 - SPARE
     MFT6 : BOOL ;	//END OF WORK MEMORY 6 - SPARE
     MFT7 : BOOL ;	//END OF WORK MEMORY 7 - SPARE
     MFT8 : BOOL ;	//END OF WORK MEMORY 8 - SPARE
    END_STRUCT ;
    SPARE : ARRAY  [1 .. 17 ] OF INT ;
   END_STRUCT ;
   C0w : STRUCT 	//PART WORD C0w
    MP : STRUCT 	//PART MEMORY / MOT PIECE
     MPP : BOOL ;	//PRESENT PART MEMORY / MEMOIRE PIECE PRESENTE
     MPAT : BOOL ;	//PART WITH WORK MEMORY / MEMOIRE PIECE A TRAVAILLER
     MPST : BOOL ;	//PART WITHOUT WORK MEMORY / MEMOIRE PIECE SANS TRAVAIL
     MPAM : BOOL ;	//PART MEMORY TO MATCH / MEMOIRE PIECE A MARIER
     MPAE : BOOL ;	//PART MEMORY TO EVACUATE / MEMOIRE PIECE A EVACUER
     MPP1 : BOOL ;	//INTERMEDIATE PRESENT PART MEMORY / MEMOIRE PIECE PRESENTE INTERMEDIAIRE
     MPP2 : BOOL ;	//INTERMEDIATE PRESENT PART MEMORY / MEMOIRE PIECE PRESENTE INTERMEDIAIRE
     MPP3 : BOOL ;	//INTERMEDIATE PRESENT PART MEMORY / MEMOIRE PIECE PRESENTE INTERMEDIAIRE
     MPP4 : BOOL ;	//INTERMEDIATE PRESENT PART MEMORY / MEMOIRE PIECE PRESENTE INTERMEDIAIRE
     MPP5 : BOOL ;	//INTERMEDIATE PRESENT PART MEMORY / MEMOIRE PIECE PRESENTE INTERMEDIAIRE
     MPP6 : BOOL ;	//INTERMEDIATE PRESENT PART MEMORY / MEMOIRE PIECE PRESENTE INTERMEDIAIRE
     MPP7 : BOOL ;	//INTERMEDIATE PRESENT PART MEMORY / MEMOIRE PIECE PRESENTE INTERMEDIAIRE
     MPP8 : BOOL ;	//INTERMEDIATE PRESENT PART MEMORY / MEMOIRE PIECE PRESENTE INTERMEDIAIRE
     MPT : BOOL ;	//PART COMPLETE MEMORY / MEMOIRE PIECE TRAVAILLE
     MPLNOK : BOOL ;	//LAUCHING PART MEMORY NOK / MEMOIRE LANCEMENT PIECE NON OK
     MPLNOR : BOOL ;	//LAUCHING PART MEMORY OK / MEMOIRE LANCEMENT PIECE OK
    END_STRUCT ;
    MS : STRUCT 	//SUPPORT WORD / MOT SUPPORT
     MSP : BOOL ;	//SUPPORT PRESENCE MEMORY / MEMOIRE SUPPORT PRESENT
     MSAE : BOOL ;	//SUPPORT TO EVACUATE MEMORY / MEMOIRE SUPPORT A EVACUER
     MSEBD : BOOL ;	//WRITING DATABASE SUPPORT MEMORY / MEMOIRE SUPPORT ECRITURE BASE DE DONNEE
     MSMBD : BOOL ;	//MODIFICATION DATABASE SUPPORT MEMORY / MEMOIRE SUPPORT MODIF BASE DE DONNEE
     MSLBD : BOOL ;	//READING DATABASE SUPPORT MEMORY / MEMOIRE SUPPORT LECTURE BASE DE DONNEE
     MSAP : BOOL ;	//PASSAGE AUTHORIZATION SUPPORT MEMORY / MEMOIRE SUPPORT AUTORISATION DE PASSAGE
     MRCPF : BOOL ;	//PART TO DO PROCESS CODE SEARCH MEMORY / MEMOIRE RECH CODES PROCESS A FAIRE
     MRCPS : BOOL ;	//NEXT PART PROCESS CODE SEARCH MEMORY / MEMOIRE RECH CODES PROCESS SUIVANT
     MSLRFID : BOOL ;	//READING RFID SUPPORT MEMORY / MEMOIRE SUPPORT LECTURE RFID
     MSERFID : BOOL ;	//WRITING RFID SUPPORT MEMORY / MEMOIRE SUPPORT ECRITURE RFID
     RES1 : BOOL ;	//SPARE / RESERVE
     RES2 : BOOL ;	//SPARE / RESERVE
     RES3 : BOOL ;	//SPARE / RESERVE
     RES4 : BOOL ;	//SPARE / RESERVE
     RES5 : BOOL ;	//SPARE / RESERVE
     RES6 : BOOL ;	//SPARE / RESERVE
    END_STRUCT ;
    NSUP : INT ;	//SUPPORT NUMBER / NUMERO DE SUPPORT
    NFILM : INT ;	//FILM NUMBER / NUMERO DE FILM
    NORDRE : INT ;	//ORDER NUMBER / NUMERO D ORDRE
    CDIV1 : INT ;	//FAMILIA / FAMILLE (CDIV1)
    CDIV2 : INT ;	//FASE / PHASE (CDIV2)
    CDIV3 : INT ;	//MODELO / MODELE (CDIV3)
    CDIV4 : INT ;	//TECHO (CDIV4)
    CDIV5 : INT ;	//VERSION (CDIV5)
    DESFI : INT ;	//FINAL DISPATCH / DESTINATION FINALE
    CSORT : INT ;	//CAUSE DE SORTIE
    DAT : STRUCT 	//DEFINITION / ATTENTE TRAVAIL
     B8 : BOOL ;	//PALETTE DE VIDAGE PERIMETRE (HORS SIPTOL)
     B9 : BOOL ;	//DEVERMINAGE PIECE / PALETTE (HORS SIPTOL)
     B10 : BOOL ;	//PALETTE DE MAP(HORS SIPTOL)
     B11 : BOOL ;	//PALETTE DE CHANGEMENT ELECTRODE BR (HORS SIPTOL)
     B12 : BOOL ;	//PALETTE DE CHANGEMENT ELECTRODE CS (HORS SIPTOL)
     B13 : BOOL ;	//DEVERMINAGE PIECE / PALETTE (AVEC SIPTOL)
     B14 : BOOL ;
     B15 : BOOL ;
     FABSPF : BOOL ;	//0 = AVEC TRAVAIL / 1 = SANS TRAVAIL (P1)
     B1 : BOOL ;
     B2 : BOOL ;	//0 = SUPPORT PLEIN / 1 = SUPPORT VIDE
     B3 : BOOL ;
     B4 : BOOL ;
     B5 : BOOL ;
     B6 : BOOL ;
     B7 : BOOL ;
    END_STRUCT ;
    CRAPI : STRUCT 	//PLC DISPATCHING REASON / CAUSE ROUTAGE API
     B8 : BOOL ;
     B9 : BOOL ;
     B10 : BOOL ;
     B11 : BOOL ;
     B12 : BOOL ;
     B13 : BOOL ;
     B14 : BOOL ;
     B15 : BOOL ;
     B0 : BOOL ;
     B1 : BOOL ;
     B2 : BOOL ;
     RARET : BOOL ;	//PIECE ANALYSE - RETOUCHE
     B4 : BOOL ;
     B5 : BOOL ;
     B6 : BOOL ;
     B7 : BOOL ;
    END_STRUCT ;
    MGEST : STRUCT 	//MOT DE GESTION RECALAGE
     MPFNOR : BOOL ;	//MEMOIRE PIECE FLUX NORMAL
     MPSTC : BOOL ;	//MEMOIRE PIECE A SORTIR TOUS CAS
     MPSOR : BOOL ;	//MEMOIRE PIECE A SORTIR (SORTIE SIPTOL BONNE)
     MPSSU : BOOL ;	//MEMOIRE PIECE A SORTIR (SUBTITUTION PIECE BONNE)
     MPSDI : BOOL ;	//MEMOIRE PIECE A SORTIR (DISCORDANCE)
     MPSSUL : BOOL ;	//MEMOIRE PIECE A SORTIR (SUBTITUTION PIECE LOUPEE)
     MPSL : BOOL ;	//MEMOIRE PIECE A SORTIR (SORTIE LOUPEE)
     MPSF99 : BOOL ;	//MEMOIRE PIECE A SORTIR (MAP FILM 99)
     MPETC : BOOL ;	//MEMOIRE PIECE A ENTRER TOUTS CAS
     MPEOR : BOOL ;	//MEMOIRE PIECE EN ENTREE (DEMANDE SIPTOL)
     MPESUB : BOOL ;	//MEMOIRE PIECE EN ENTREE (SUBTITUTION PIECE BONNE)
     MPEDI : BOOL ;	//MEMOIRE PIECE EN ENTREE (DISCORDANCE)
     MPESUL : BOOL ;	//MEMOIRE PIECE EN ENTREE (SUBTITUTION PIECE LOUPEE)
     MPOCV : BOOL ;	//MEMOIRE PIECE A SORTIR VEHICULE ANNULE + CROCHET VIDE
     MESUTC : BOOL ;	//MEMOIRE EN ENTREE SUBSTITUTION TOUS CAS (PIECE BONNE OU MAUVAISE)
     MSSUTC : BOOL ;	//MEMOIRE SORTIE SUBSTITUTION TOUS CAS (PIECE BONNE OU MAUVAISE)
    END_STRUCT ;
    TVEH : STRUCT 	//TYPO DE VEHICULO
     B8 : BOOL ;
     B9 : BOOL ;
     B10 : BOOL ;
     B11 : BOOL ;
     B12 : BOOL ;
     B13 : BOOL ;
     B14 : BOOL ;
     FABSPF : BOOL ;	//FABRICATION SANS PIECE AU FILM
     SPE : BOOL ;	//UNIT ESPECIAL
     B1 : BOOL ;
     B2 : BOOL ;
     B3 : BOOL ;
     B4 : BOOL ;
     B5 : BOOL ;
     B6 : BOOL ;
     B7 : BOOL ;
    END_STRUCT ;
    SPARE : ARRAY  [1 .. 4 ] OF INT ;
   END_STRUCT ;
  END_STRUCT ;	
BEGIN
END_DATA_BLOCK

ORGANIZATION_BLOCK OB 1
TITLE = "Main Program Sweep (Cycle)"
VERSION : 0.1
VAR_TEMP
  OB1_EV_CLASS : BYTE ;	//Bits 0-3 = 1 (Coming event), Bits 4-7 = 1 (Event class 1)
  OB1_SCAN_1 : BYTE ;	//1 (Cold restart scan 1 of OB 1), 3 (Scan 2-n of OB 1)
  OB1_PRIORITY : BYTE ;	//Priority of OB Execution
  OB1_OB_NUMBR : BYTE ;	//1 (Organization block 1, OB1)
  OB1_RESERVED_1 : BYTE ;	//Reserved for system
  OB1_RESERVED_2 : BYTE ;	//Reserved for system
  OB1_PREV_CYCLE : INT ;	//Cycle time of previous OB1 scan (milliseconds)
  OB1_MIN_CYCLE : INT ;	//Minimum cycle time of OB1 (milliseconds)
  OB1_MAX_CYCLE : INT ;	//Maximum cycle time of OB1 (milliseconds)
  OB1_DATE_TIME : DATE_AND_TIME ;	//Date and time OB1 started
END_VAR
BEGIN
// (block stored without names or comments; labels and parameter names are numbered)
END_ORGANIZATION_BLOCK

